	IF xStFct_SetForceDeflection THEN
		IF NOT(xStFct_InitSetForceDeflection) THEN
			IF NOT(ptrTCylToolDeflection^.T_CtrleCyl.xExecute) AND ptrTCylToolDeflection^.T_CtrleCyl.xDone THEN
				xStFct_InitSetForceDeflection:=TRUE;
				ptrTCylToolDeflection^.T_CtrleCyl.iFunction:=4;
				ptrTCylToolDeflection^.T_CtrleCyl.xExecute:=TRUE;
			END_IF;
		END_IF;
		IF NOT(ptrTCylToolDeflection^.T_CtrleCyl.xExecute) AND ptrTCylToolDeflection^.T_CtrleCyl.xDone AND xStFct_InitSetForceDeflection THEN
			xStFct_InitSetForceDeflection:=FALSE;
			xStFct_SetForceDeflection:=FALSE;
		END_IF;
	END_IF;
END_IF;
END_ACTION
ACTION StationFunction_Ctrl_Stop:
IF xStFct_TmpStop AND NOT(xStFct_SetEnd) THEN
	CASE iStFct_TmpStopStep OF
		1:	IF gxHardwareOFF OR gxAxisOFF THEN
				iStFct_TmpStopStep:=9;
				RETURN;
			END_IF;
			IF (NOT(ptrTAxisZ^.T_CtrleSingle.xNotMoving) OR NOT(ptrTAxisZ^.T_CtrleSingle.xDone)) AND
			     NOT((ptrTAxisZ^.T_CtrleSingle.iFunction = 5) AND NOT(ptrTAxisZ^.T_CtrleSingle.xDone)) THEN
				ptrTAxisZ^.T_CtrleSingle.iFunction:=5;
				ptrTAxisZ^.T_CtrleSingle.xExecute:=TRUE;
			END_IF;
			IF (iStationFunctionNr = 5) AND ((iStFct_StepPrc = 3) OR (iStFct_StepPrc = 40)) THEN
				IF (T_Station_Parameter.T_StProcess.iWorkControlType > 1) THEN
					T_Z_St1_Ctrle.diVelocityCommandValue:=0;
					gxZAxisVelocityCtrlActive:=TRUE;
					ptrTAxisZ^.T_CtrleSingle.iFunction:=5;
					ptrTAxisZ^.T_CtrleSingle.xExecute:=TRUE;
				END_IF;
			END_IF;
			IF (NOT(ptrTAxisS^.T_CtrleSingle.xNotMoving) OR NOT(ptrTAxisS^.T_CtrleSingle.xDone)) AND
			     NOT((ptrTAxisS^.T_CtrleSingle.iFunction = 5) AND NOT(ptrTAxisS^.T_CtrleSingle.xDone)) THEN
				ptrTAxisS^.T_CtrleSingle.iFunction:=5;
				ptrTAxisS^.T_CtrleSingle.xExecute:=TRUE;
			END_IF;
			iStFct_TmpStopStep:=iStFct_TmpStopStep + 1;
			T_Station_Work.TCtrlOnlineChange.xLockChange_Z_WorkSpeedForward:=TRUE;
			T_Station_Work.TCtrlOnlineChange.xLockChange_Z_WorkSpeedBackward:=TRUE;
			QxCoolant_St1:=FALSE;
			QxFastStrokeOn_St1:=FALSE;
		2:	IF ptrTAxisZ^.T_CtrleSingle.xNotMoving AND ptrTAxisS^.T_CtrleSingle.xNotMoving AND NOT(gxZAxisVelocityCtrlActive) THEN
				iStFct_TmpStopStep:=iStFct_TmpStopStep + 1;
			ELSE
				IF NOT(gxZAxisVelocityCtrlActive) THEN
					iStFct_TmpStopStep:=1;
				ELSE
					iStFct_TmpStopStep:=10;
				END_IF;
			END_IF;
		3:	IF TRUE THEN
				IF (iStationFunctionNr = 4) OR (iStationFunctionNr = 5) THEN
					iStFct_TmpStopStep:=iStFct_TmpStopStep + 1;
				ELSE
					iStFct_TmpStopStep:=iStFct_TmpStopStep + 6;
				END_IF;
			END_IF;
		4:	T_Station_Work.THWWorkStation.TCtrlWork.xWorkingFinished:=TRUE;
			IF (T_Station_Work.THWWorkStation.TCtrlWork.bPartQuality = 7) THEN
				T_Station_Work.THWWorkStation.TCtrlWork.bPartQuality:=8;	(* < Bearb. abgbr. > *)
			END_IF;
			ptrTAxisZ^.T_CtrleSingle.iFunction:=7;	(* Absolut Bewegung *)
			ptrTAxisZ^.T_CtrleSingle.lrPosition:=grZ_LoadPos;	(* AxisSlide auf LadePosition setzen *)
			ptrTAxisZ^.T_CtrleSingle.lrVelocity:=rOutfeedStrokeAxisSpeed;
			ptrTAxisZ^.T_CtrleSingle.xExecute:=TRUE;
			(* Spindel mit Ausfahrgeschwindigkeit *)
			IF ptrTAxisS^.T_CtrleSingle.xNotMoving THEN
				ptrTAxisS^.T_CtrleSingle.iFunction:=6;	(* Move Velocity *)
			ELSE
				ptrTAxisS^.T_CtrleSingle.iFunction:=12;	(* Move Velocity *)
			END_IF;
			ptrTAxisS^.T_CtrleSingle.lrVelocity:=T_Station_Parameter.T_StProcess.rOutfeedSpindleSpeed;
			ptrTAxisS^.T_CtrleSingle.xExecute:=TRUE;
			IF NOT(ptrTAxisBubbler^.T_CtrleDCAxis.xNotMoving) THEN
				(* Abstreifer ZU *)
				QxCylStripperClose_St1:=TRUE;
				QxCylStripperOpen_St1:=FALSE;
			END_IF
			iStFct_TmpStopStep:=iStFct_TmpStopStep + 1;
		5:	IF NOT(ptrTAxisZ^.T_CtrleSingle.xExecute) AND ptrTAxisZ^.T_CtrleSingle.xDone AND
			     NOT(ptrTAxisS^.T_CtrleSingle.xExecute) AND ptrTAxisS^.T_CtrleSingle.xDone THEN
				iStFct_TmpStopStep:=iStFct_TmpStopStep + 1;
			END_IF;
		6:	IF TRUE THEN
				iStFct_TmpStopStep:=iStFct_TmpStopStep + 1;
			END_IF;
		7:	iStFct_TmpStopStep:=iStFct_TmpStopStep + 1;
		8:	IF NOT(ptrTAxisZ^.T_CtrleSingle.xExecute) AND ptrTAxisZ^.T_CtrleSingle.xDone THEN
				iStFct_TmpStopStep:=iStFct_TmpStopStep + 1;
			END_IF;
		9:	IF TRUE THEN
				xStFct_TmpStop:=FALSE;
				iStFct_TmpStopStep:=1;
				xStFct_SetEnd:=TRUE;
				(* Abstreifer AUF *)
				QxCylStripperClose_St1:=FALSE;
				QxCylStripperOpen_St1:=TRUE;
				QxCylWPUnfix_St1:=FALSE;
				gxSuspensionONOFF:=FALSE;
			END_IF;
		10:	IF NOT(ptrTAxisZ^.T_CtrleSingle.xExecute) AND ptrTAxisZ^.T_CtrleSingle.xDone AND ptrTAxisS^.T_CtrleSingle.xNotMoving THEN
				gxZAxisVelocityCtrlActive:=FALSE;
				iStFct_TmpStopStep:=3;
			END_IF;
	END_CASE;
END_IF;
END_ACTION
ACTION StationFunction_Ctrl_ToolSpindle:
IF NOT(xSafetyCircuitOn) THEN
	T_Station_Work.THWWorkStation.TCtrlWork.xWorkStartToolRotation:=FALSE;
	T_Station_Work.THWWorkStation.TCtrlWork.xWorkStopToolRotation:=FALSE;
END_IF;
IF T_Station_Work.THWWorkStation.TCtrlWork.xWorkStartToolRotation AND NOT(T_Station_Work.THWWorkStation.TCtrlWork.xWorkStopToolRotation) THEN
	CASE iStFct_StepStartToolSpindle OF
	1:	IF NOT(xStFct_InitStepStartToolSpindle) THEN
			IF NOT(ptrTAxisS^.T_CtrleSingle.xExecute) AND NOT(ptrTAxisS^.T_CtrleSingle.xPower) AND ptrTAxisS^.T_CtrleSingle.xDone THEN
				xStFct_InitStepStartToolSpindle:=TRUE;
				ptrTAxisS^.T_CtrleSingle.iFunction:=3;	(* Strom einschalten *)
				ptrTAxisS^.T_CtrleSingle.xExecute:=TRUE;
			END_IF;
		END_IF;
		IF NOT(ptrTAxisS^.T_CtrleSingle.xExecute) AND ptrTAxisS^.T_CtrleSingle.xDone AND ptrTAxisS^.T_CtrleSingle.xPower THEN
			xStFct_InitStepStartToolSpindle:=FALSE;
			iStFct_StepStartToolSpindle:=iStFct_StepStartToolSpindle + 1;
		END_IF;
	2:	IF NOT(xStFct_InitStepStartToolSpindle) THEN
			xStFct_InitStepStartToolSpindle:=TRUE;
			(* Neu-->Hier wird die Spindel nicht mehr mittels der Einfädelgeschwindigkeit gestartet, sondern nur direkt über die Stationseinfädelfunktion *)
		END_IF;
		IF NOT(ptrTAxisS^.T_CtrleSingle.xExecute) AND ptrTAxisS^.T_CtrleSingle.xDone THEN
			xStFct_InitStepStartToolSpindle:=FALSE;
			iStFct_StepStartToolSpindle:=iStFct_StepStartToolSpindle + 1;
		END_IF;
	(* Abwarten bis Einfädeln Bearbeitungsfunktion gestartet hat *)
	3:	IF xStartFunction AND (iStationFunctionNr = 4) THEN
			xStFct_InitStepStartToolSpindle:=FALSE;
			iStFct_StepStartToolSpindle:=iStFct_StepStartToolSpindle + 1;
		END_IF;
	(* Abwarten bis Bearbeitungsfunktion beendet hat *)
	4:	IF NOT(xStartFunction) AND (iStationFunctionNr = 5) THEN
			xStFct_InitStepStartToolSpindle:=FALSE;
			iStFct_StepStartToolSpindle:=iStFct_StepStartToolSpindle + 1;	(* Neu-->Spindel wird gestoppt, und dann erst wieder gestartet direkt über die Stationseinfädelfunktion *)
		END_IF;
	5:	IF NOT(xStFct_InitStepStartToolSpindle) THEN
			IF NOT(ptrTAxisS^.T_CtrleSingle.xExecute) AND NOT(ptrTAxisS^.T_CtrleSingle.xNotMoving) AND
			     ptrTAxisS^.T_CtrleSingle.xDone AND (ptrTAxisS^.T_CtrleSingle.iFunction <> 5) THEN
				xStFct_InitStepStartToolSpindle:=TRUE;
				ptrTAxisS^.T_CtrleSingle.iFunction:=5;	(* Rotation stoppen *)
				ptrTAxisS^.T_CtrleSingle.xExecute:=TRUE;
			END_IF;
		END_IF;
		IF NOT(ptrTAxisS^.T_CtrleSingle.xExecute) AND ptrTAxisS^.T_CtrleSingle.xDone AND ptrTAxisS^.T_CtrleSingle.xNotMoving THEN
			xStFct_InitStepStartToolSpindle:=FALSE;
			iStFct_StepStartToolSpindle:=1;
		ELSE
			xStFct_InitStepStartToolSpindle:=FALSE;
		END_IF;
	END_CASE;
ELSE
	iStFct_StepStartToolSpindle:=1;
	xStFct_InitStepStartToolSpindle:=FALSE;
END_IF;
IF T_Station_Work.THWWorkStation.TCtrlWork.xWorkStopToolRotation THEN
	T_Station_Work.THWWorkStation.TCtrlWork.xWorkStartToolRotation:=FALSE;
	CASE iStFct_StepStopToolSpindle OF
	1:	IF NOT(xStFct_InitStepStopToolSpindle) THEN
			IF NOT(ptrTAxisS^.T_CtrleSingle.xExecute) AND NOT(ptrTAxisS^.T_CtrleSingle.xNotMoving) AND
			     ptrTAxisS^.T_CtrleSingle.xDone AND (ptrTAxisS^.T_CtrleSingle.iFunction <> 5) THEN
				xStFct_InitStepStopToolSpindle:=TRUE;
				ptrTAxisS^.T_CtrleSingle.iFunction:=5;	(* Rotation stoppen *)
				ptrTAxisS^.T_CtrleSingle.xExecute:=TRUE;
			END_IF;
		END_IF;
		IF NOT(ptrTAxisS^.T_CtrleSingle.xExecute) AND ptrTAxisS^.T_CtrleSingle.xDone AND ptrTAxisS^.T_CtrleSingle.xNotMoving THEN
			xStFct_InitStepStopToolSpindle:=FALSE;
			iStFct_StepStopToolSpindle:=iStFct_StepStopToolSpindle + 1;
		ELSE
			xStFct_InitStepStopToolSpindle:=FALSE;
		END_IF;
	2:	IF NOT(xStFct_InitStepStopToolSpindle) THEN
			IF NOT(ptrTAxisS^.T_CtrleSingle.xExecute) AND ptrTAxisS^.T_CtrleSingle.xPower AND ptrTAxisS^.T_CtrleSingle.xDone THEN
				xStFct_InitStepStopToolSpindle:=TRUE;
				ptrTAxisS^.T_CtrleSingle.iFunction:=4;	(* Stromlos schalten *)
				ptrTAxisS^.T_CtrleSingle.xExecute:=TRUE;
			END_IF;
		END_IF;
		IF NOT(ptrTAxisS^.T_CtrleSingle.xExecute) AND ptrTAxisS^.T_CtrleSingle.xDone AND NOT(ptrTAxisS^.T_CtrleSingle.xPower) THEN
			xStFct_InitStepStopToolSpindle:=FALSE;
			iStFct_StepStopToolSpindle:=1;
			T_Station_Work.THWWorkStation.TCtrlWork.xWorkStopToolRotation:=FALSE;
		END_IF;
		IF NOT(ptrTAxisS^.T_CtrleSingle.xExecute) AND NOT(ptrTAxisS^.T_CtrleSingle.xNotMoving) THEN
			xStFct_InitStepStopToolSpindle:=FALSE;
			iStFct_StepStopToolSpindle:=1;
		END_IF;
	END_CASE;
ELSE
	iStFct_StepStopToolSpindle:=1;
	xStFct_InitStepStopToolSpindle:=FALSE;
END_IF;
END_ACTION
ACTION StationFunction_Fct_01_Referencing:
(******************************************************************************************************************************************)
(****************************				           Reset Stationsfunktion                                            *****************************)
(******************************************************************************************************************************************)
StationFunction_Ctrl_Reset;
(******************************************************************************************************************************************)
(****************************			        Stationsfunktion Fehler Controller                                    *****************************)
(******************************************************************************************************************************************)
StationFunction_Ctrl_Error;
(******************************************************************************************************************************************)
(****************************				    Stationsfunktion Haupt Controller                               *****************************)
(******************************************************************************************************************************************)
StationFunction_Ctrl_Main;
(******************************************************************************************************************************************)
(****************************			         Stationsfunktion sofort Unterbrechung                           *****************************)
(******************************************************************************************************************************************)
StationFunction_Ctrl_Stop;
(******************************************************************************************************************************************)
(****************************			             Stationsfunktion Hauptablauf                                       *****************************)
(******************************************************************************************************************************************)
IF xStFct_StartMainPrc AND NOT(xStFct_SetEnd) AND NOT(xStFct_HardwareError) AND NOT(xStFct_TmpStop) THEN
	CASE iStFct_StepPrc OF
	1:	xStFct_StartMainPrc:=FALSE;
		xStFct_InitStep:=FALSE;
		iStFct_StepPrc:=1;
	END_CASE;
END_IF;
(******************************************************************************************************************************************)
(****************************			             Stationsfunktion Parallelablauf                                       *****************************)
(******************************************************************************************************************************************)
IF xStFct_StartPrc_Parallel AND NOT(xStFct_SetEnd) AND NOT(xStFct_HardwareError) THEN
	CASE iStFct_StepPrc_Parallel OF
	1:	iStFct_StepPrc_Parallel:=1;
		xStFct_InitStep_Parallel:=FALSE;
		xStFct_StartPrc_Parallel:=FALSE;
	END_CASE;
END_IF;
(******************************************************************************************************************************************)
(****************************				     Stationsfunktion Endprozedur                                    *****************************)
(******************************************************************************************************************************************)
StationFunction_Ctrl_End;
END_ACTION
ACTION StationFunction_Fct_02_InitialState:
(******************************************************************************************************************************************)
(****************************				           Reset Stationsfunktion                                            *****************************)
(******************************************************************************************************************************************)
StationFunction_Ctrl_Reset;
(******************************************************************************************************************************************)
(****************************			        Stationsfunktion Fehler Controller                                    *****************************)
(******************************************************************************************************************************************)
StationFunction_Ctrl_Error;
(******************************************************************************************************************************************)
(****************************				    Stationsfunktion Haupt Controller                               *****************************)
(******************************************************************************************************************************************)
StationFunction_Ctrl_Main;
(******************************************************************************************************************************************)
(****************************			         Stationsfunktion sofort Unterbrechung                           *****************************)
(******************************************************************************************************************************************)
StationFunction_Ctrl_Stop;
(******************************************************************************************************************************************)
(****************************			             Stationsfunktion Hauptablauf                                       *****************************)
(******************************************************************************************************************************************)
IF xStFct_StartMainPrc AND NOT(xStFct_SetEnd) AND NOT(xStFct_HardwareError) AND NOT(xStFct_TmpStop) THEN
(***************************************************************************************************************************************************)
	CASE iStFct_StepPrc OF
	1:	wStFct_Status:=0;
		xBlockCheckLimitSwitch:=TRUE;
		IF gxHardwareOFF OR gxAxisOFF THEN
			iStFct_StepPrc:=12;
			RETURN;
		END_IF;
		IF NOT(ptrTAxisZ^.T_CtrleSingle.xRef) THEN	(* Z Achse muss referenziert sein *)
			xStFct_HardwareError:=TRUE;
			diStFct_TmpErrorNr:=12;	(* Z Achse muss referenziert sein *)
			RETURN;
		END_IF;
		(* Überprüfe alle Positionen der Z Achse *)
		StationFunction_Ctrl_CheckPos_Z;
		IF xStFct_PositionOutRange_Z THEN
			xStFct_HardwareError:=TRUE;
			diStFct_TmpErrorNr:=iStFct_PosErrorNr;
			RETURN;
		END_IF;
		IF NOT(xStFct_InitStep) THEN
			(* Falls Z Achse sich bewegt, dann wird der Motor gestoppt *)
			IF NOT(ptrTAxisZ^.T_CtrleSingle.xExecute) AND NOT(ptrTAxisZ^.T_CtrleSingle.xNotMoving) THEN
				xStFct_InitStep:=TRUE;
				ptrTAxisZ^.T_CtrleSingle.iFunction:=5;
				ptrTAxisZ^.T_CtrleSingle.xExecute:=TRUE;
			END_IF;
		END_IF;
		IF NOT(ptrTAxisZ^.T_CtrleSingle.xExecute) AND ptrTAxisZ^.T_CtrleSingle.xDone AND ptrTAxisZ^.T_CtrleSingle.xNotMoving THEN
			xStFct_StartMainPrc:=FALSE;
			xStFct_InitStep:=FALSE;
			iStFct_StepPrc:=iStFct_StepPrc + 1;
		END_IF;
	2:	IF NOT(xStFct_InitStep) THEN
			(* Falls Z Achse nicht bestromt ist, dann wird der Motorstrom eingeschaltet *)
			IF NOT(ptrTAxisZ^.T_CtrleSingle.xPower) THEN
				xStFct_InitStep:=TRUE;
				ptrTAxisZ^.T_CtrleSingle.iFunction:=3;	(* Strom einschalten *)
				ptrTAxisZ^.T_CtrleSingle.xExecute:=TRUE;
			END_IF;
			QxCylStripperClose_St1:=FALSE;
			QxCylStripperOpen_St1:=TRUE;
			QxCylWPUnfix_St1:=FALSE;
			gxSuspensionONOFF:=FALSE;
		END_IF;
		IF NOT(ptrTAxisZ^.T_CtrleSingle.xExecute) AND ptrTAxisZ^.T_CtrleSingle.xDone AND ptrTAxisZ^.T_CtrleSingle.xPower THEN
			xStFct_StartMainPrc:=FALSE;
			xStFct_InitStep:=FALSE;
			iStFct_StepPrc:=iStFct_StepPrc + 1;
		END_IF;
	3:	IF NOT(xStFct_InitStep) THEN
			xStFct_InitStep:=TRUE;
			(* Zylinder für Auslenkung-->mit Workauslenkkraft *)
			ptrTCylToolDeflection^.T_CtrleCyl.iFunction:=2;
			ptrTCylToolDeflection^.T_Config.tDelayOn:=T#0.4s;
			ptrTCylToolDeflection^.T_CtrleCyl.T_Analog.rForceIn:=T_Station_Parameter.T_OnlineChange.rForceDeflection;
			ptrTCylToolDeflection^.T_CtrleCyl.xExecute:=TRUE;
			(* Zylinder für Drehmoment HC-->mit Schwellwert Startposition *)
			ptrTCylToolTorqueHC^.T_CtrleCyl.iFunction:=2;
			ptrTCylToolTorqueHC^.T_Config.tDelayOn:=T#0.2s;
			ptrTCylToolTorqueHC^.T_CtrleCyl.T_Analog.rForceIn:=T_Station_Parameter.T_OnlineChange.rTorqueLevelHC;
			ptrTCylToolTorqueHC^.T_CtrleCyl.xExecute:=TRUE;
			(* Zylinder für Überlast Drehmoment *)
			ptrTCylToolTorqueOverload^.T_CtrleCyl.iFunction:=2;
			ptrTCylToolTorqueOverload^.T_Config.tDelayOn:=T#0.2s;
			ptrTCylToolTorqueOverload^.T_CtrleCyl.T_Analog.rForceIn:=T_Station_Parameter.T_StProcess.rTorqueLevel_Overload;
			ptrTCylToolTorqueOverload^.T_CtrleCyl.xExecute:=TRUE;
		END_IF;
		IF NOT(ptrTCylToolDeflection^.T_CtrleCyl.xExecute) AND ptrTCylToolDeflection^.T_CtrleCyl.xDone AND
		    NOT(ptrTCylToolTorqueHC^.T_CtrleCyl.xExecute) AND ptrTCylToolTorqueHC^.T_CtrleCyl.xDone AND
		    NOT(ptrTCylToolTorqueOverload^.T_CtrleCyl.xExecute) AND ptrTCylToolTorqueOverload^.T_CtrleCyl.xDone THEN
			xStFct_StartMainPrc:=FALSE;
			xStFct_InitStep:=FALSE;
			IF NOT(ptrTAxisZ^.T_CtrleSingle.xStateHWLimitNeg) AND NOT(ptrTAxisZ^.T_CtrleSingle.xStateHWLimitPos) THEN
				iStFct_StepPrc:=iStFct_StepPrc + 4;
			ELSE
				IF ptrTAxisZ^.T_CtrleSingle.xStateHWLimitNeg AND ptrTAxisZ^.T_CtrleSingle.xStateHWLimitPos THEN
					xStFct_HardwareError:=TRUE;
					diStFct_TmpErrorNr:=3;	(* Z Achse-->Positiver + Negativer HW Endschalter Aktiv *)
					RETURN;
				ELSIF ptrTAxisZ^.T_CtrleSingle.xStateHWLimitNeg THEN
					iStFct_StepPrc:=iStFct_StepPrc + 1;
				ELSE
					iStFct_StepPrc:=iStFct_StepPrc + 2;
				END_IF;
			END_IF;
		END_IF;
	(* Wegfahren vom negativen Endschalters *)
	4:	IF NOT(xStFct_InitStep) THEN
			xStFct_InitStep:=TRUE;
			ptrTAxisZ^.T_CtrleSingle.iFunction:=6;	(* Geschwindigkeits Bewegung *)
			ptrTAxisZ^.T_CtrleSingle.lrVelocity:=1.0;
			ptrTAxisZ^.T_CtrleSingle.xExecute:=TRUE;
		END_IF;
		IF NOT(ptrTAxisZ^.T_CtrleSingle.xStateHWLimitNeg) THEN
			xStFct_StartMainPrc:=FALSE;
			xStFct_InitStep:=FALSE;
			iStFct_StepPrc:=iStFct_StepPrc + 2;
		END_IF;
		IF ptrTAxisZ^.T_CtrleSingle.xStateHWLimitNeg AND ptrTAxisZ^.T_CtrleSingle.xStateHWLimitPos THEN
			xStFct_HardwareError:=TRUE;
			diStFct_TmpErrorNr:=3;	(* Z Achse-->Positiver + Negativer HW Endschalter Aktiv *)
		END_IF;
	(* Wegfahren vom positiven Endschalters *)
	5:	IF NOT(xStFct_InitStep) THEN
			xStFct_InitStep:=TRUE;
			ptrTAxisZ^.T_CtrleSingle.iFunction:=6;	(* Geschwindigkeits Bewegung *)
			ptrTAxisZ^.T_CtrleSingle.lrVelocity:=-1.0;
			ptrTAxisZ^.T_CtrleSingle.xExecute:=TRUE;
		END_IF;
		IF NOT(ptrTAxisZ^.T_CtrleSingle.xStateHWLimitPos) THEN
			xStFct_StartMainPrc:=FALSE;
			xStFct_InitStep:=FALSE;
			iStFct_StepPrc:=iStFct_StepPrc + 1;
		END_IF;
		IF ptrTAxisZ^.T_CtrleSingle.xStateHWLimitNeg AND ptrTAxisZ^.T_CtrleSingle.xStateHWLimitPos THEN
			xStFct_HardwareError:=TRUE;
			diStFct_TmpErrorNr:=3;	(* Z Achse-->Positiver + Negativer HW Endschalter Aktiv *)
		END_IF;
	(* Stoppen der Bewegung *)
	6:	IF NOT(xStFct_InitStep) THEN
			xStFct_InitStep:=TRUE;
			ptrTAxisZ^.T_CtrleSingle.iFunction:=5;
			ptrTAxisZ^.T_CtrleSingle.xExecute:=TRUE;
		END_IF;
		IF NOT(ptrTAxisZ^.T_CtrleSingle.xExecute) AND ptrTAxisZ^.T_CtrleSingle.xDone THEN
			xStFct_StartMainPrc:=FALSE;
			xStFct_InitStep:=FALSE;
			iStFct_StepPrc:=iStFct_StepPrc + 1;
		END_IF;
	(* Aktuatoren in Ausgangslage bringen *)
	7:	IF NOT(xStFct_InitStep) THEN
			xStFct_InitStep:=TRUE;
			xBlockCheckLimitSwitch:=FALSE;
		END_IF;
		IF TRUE THEN
			xStFct_StartMainPrc:=FALSE;
			xStFct_InitStep:=FALSE;
			iStFct_StepPrc:=iStFct_StepPrc + 1;
		END_IF;
	8:	IF NOT(xStFct_InitStep) THEN
			xStFct_InitStep:=TRUE;
			IF (ptrTAxisZ^.T_LiveValue.lrActualPosition > grZ_LoadPos) THEN
				ptrTAxisZ^.T_CtrleSingle.iFunction:=7;	(* Absolut Bewegung *)
				ptrTAxisZ^.T_CtrleSingle.lrPosition:=grZ_LoadPos;	(* AxisSlide auf LadePosition setzen *)
				ptrTAxisZ^.T_CtrleSingle.lrVelocity:=T_Station_Parameter.T_StProcess.rOutfeedStrokeAxisSpeed;
				ptrTAxisZ^.T_CtrleSingle.xExecute:=TRUE;
			END_IF;
		END_IF;
		IF NOT(ptrTAxisZ^.T_CtrleSingle.xExecute) AND ptrTAxisZ^.T_CtrleSingle.xDone THEN
			xStFct_StartMainPrc:=FALSE;
			xStFct_InitStep:=FALSE;
			iStFct_StepPrc:=iStFct_StepPrc + 1;
		END_IF;
	(* Aktuatoren in Ausgangslage bringen *)
	9:	IF NOT(xStFct_InitStep) THEN
			xStFct_InitStep:=TRUE;
		END_IF;
		IF NOT(ptrTAxisZ^.T_CtrleSingle.xExecute) AND ptrTAxisZ^.T_CtrleSingle.xDone THEN
			xStFct_StartMainPrc:=FALSE;
			xStFct_InitStep:=FALSE;
			iStFct_StepPrc:=iStFct_StepPrc + 1;
		END_IF;
	(* Aktuatoren in Ausgangslage bringen *)
	10:	IF NOT(xStFct_InitStep) THEN
			xStFct_InitStep:=TRUE;
		END_IF;
		IF NOT(ptrTAxisZ^.T_CtrleSingle.xExecute) AND ptrTAxisZ^.T_CtrleSingle.xDone THEN
			xStFct_StartMainPrc:=FALSE;
			xStFct_InitStep:=FALSE;
			iStFct_StepPrc:=iStFct_StepPrc + 1;
		END_IF;
	11:	IF NOT(xStFct_InitStep) THEN
			xStFct_InitStep:=TRUE;
		END_IF;
		IF NOT(ptrTAxisZ^.T_CtrleSingle.xExecute) AND ptrTAxisZ^.T_CtrleSingle.xDone THEN
			xStFct_StartMainPrc:=FALSE;
			xStFct_InitStep:=FALSE;
			iStFct_StepPrc:=iStFct_StepPrc + 1;
		END_IF;
	12:	xStFct_StartMainPrc:=FALSE;
		xStFct_InitStep:=FALSE;
		iStFct_StepPrc:=0;
		xStFct_SetEnd:=TRUE;
	END_CASE;
END_IF;
(******************************************************************************************************************************************)
(****************************			             Stationsfunktion Parallelablauf                                       *****************************)
(******************************************************************************************************************************************)
IF xStFct_StartPrc_Parallel AND NOT(xStFct_SetEnd) AND NOT(xStFct_HardwareError) THEN
	CASE iStFct_StepPrc_Parallel OF
	1:	iStFct_StepPrc_Parallel:=1;
		xStFct_InitStep_Parallel:=FALSE;
		xStFct_StartPrc_Parallel:=FALSE;
	END_CASE;
END_IF;
(******************************************************************************************************************************************)
(****************************				     Stationsfunktion Endprozedur                                    *****************************)
(******************************************************************************************************************************************)
StationFunction_Ctrl_End;
END_ACTION
ACTION StationFunction_Fct_03_ToolRotationON:
;(******************************************************************************************************************************************)
(****************************				           Reset Stationsfunktion                                            *****************************)
(******************************************************************************************************************************************)
StationFunction_Ctrl_Reset;
(******************************************************************************************************************************************)
(****************************			        Stationsfunktion Fehler Controller                                    *****************************)
(******************************************************************************************************************************************)
StationFunction_Ctrl_Error;
(******************************************************************************************************************************************)
(****************************				    Stationsfunktion Haupt Controller                               *****************************)
(******************************************************************************************************************************************)
StationFunction_Ctrl_Main;
(******************************************************************************************************************************************)
(****************************			         Stationsfunktion sofort Unterbrechung                           *****************************)
(******************************************************************************************************************************************)
StationFunction_Ctrl_Stop;
(******************************************************************************************************************************************)
(****************************			             Stationsfunktion Hauptablauf                                       *****************************)
(******************************************************************************************************************************************)
IF xStFct_StartMainPrc AND NOT(xStFct_SetEnd) AND NOT(xStFct_HardwareError) AND NOT(xStFct_TmpStop) THEN
	IF T_Station_Work.THWWorkStation.TCtrlWork.xWorkStopToolRotation THEN
		xStFct_StartMainPrc:=FALSE;
		xStFct_InitStep:=FALSE;
		iStFct_StepPrc:=0;
		xStFct_SetEnd:=TRUE;
	END_IF;
	CASE iStFct_StepPrc OF
	1:	IF NOT(xStFct_InitStep) THEN
			(* Falls die Spindel nicht bestromt ist, dann wird der Motorstrom eingeschaltet *)
			IF NOT(ptrTAxisS^.T_CtrleSingle.xPower) THEN
				xStFct_InitStep:=TRUE;
				ptrTAxisS^.T_CtrleSingle.iFunction:=3;	(* Strom einschalten *)
				ptrTAxisS^.T_CtrleSingle.xExecute:=TRUE;
			END_IF;
		END_IF;
		IF NOT(ptrTAxisS^.T_CtrleSingle.xExecute) AND ptrTAxisS^.T_CtrleSingle.xDone AND ptrTAxisS^.T_CtrleSingle.xPower THEN
			xStFct_StartMainPrc:=FALSE;
			xStFct_InitStep:=FALSE;
			iStFct_StepPrc:=iStFct_StepPrc + 1;
		END_IF;
	2:	IF NOT(xStFct_InitStep) THEN
			xStFct_InitStep:=TRUE;
			(* Zylinder für Auslenkung-->mit Workauslenkkraft *)
			ptrTCylToolDeflection^.T_CtrleCyl.iFunction:=2;
			ptrTCylToolDeflection^.T_Config.tDelayOn:=T#0.3s;
			ptrTCylToolDeflection^.T_CtrleCyl.T_Analog.rForceIn:=T_Station_Parameter.T_OnlineChange.rForceDeflection;
			ptrTCylToolDeflection^.T_CtrleCyl.xExecute:=TRUE;
			(* Zylinder für Drehmoment HC-->mit Schwellwert Startposition *)
			ptrTCylToolTorqueHC^.T_CtrleCyl.iFunction:=2;
			ptrTCylToolTorqueHC^.T_Config.tDelayOn:=T#0.2s;
			ptrTCylToolTorqueHC^.T_CtrleCyl.T_Analog.rForceIn:=T_Station_Parameter.T_OnlineChange.rTorqueLevelHC;
			ptrTCylToolTorqueHC^.T_CtrleCyl.xExecute:=TRUE;
			(* Zylinder für Überlast Drehmoment *)
			ptrTCylToolTorqueOverload^.T_CtrleCyl.iFunction:=2;
			ptrTCylToolTorqueOverload^.T_Config.tDelayOn:=T#0.2s;
			ptrTCylToolTorqueOverload^.T_CtrleCyl.T_Analog.rForceIn:=T_Station_Parameter.T_StProcess.rTorqueLevel_Overload;
			ptrTCylToolTorqueOverload^.T_CtrleCyl.xExecute:=TRUE;
			IF ptrTAxisS^.T_CtrleSingle.xNotMoving THEN
				ptrTAxisS^.T_CtrleSingle.iFunction:=6;	(* Move Velocity *)
			ELSE
				ptrTAxisS^.T_CtrleSingle.iFunction:=12;	(* Move Velocity with new velocity *)
			END_IF;
			ptrTAxisS^.T_CtrleSingle.lrVelocity:=T_Station_Parameter.T_OnlineChange.rWorkingSpindleSpeed;
			ptrTAxisS^.T_CtrleSingle.xExecute:=TRUE;
		END_IF;
		IF NOT(ptrTCylToolDeflection^.T_CtrleCyl.xExecute) AND ptrTCylToolDeflection^.T_CtrleCyl.xDone AND
		     NOT(ptrTCylToolTorqueHC^.T_CtrleCyl.xExecute) AND ptrTCylToolTorqueHC^.T_CtrleCyl.xDone AND
		     NOT(ptrTCylToolTorqueOverload^.T_CtrleCyl.xExecute) AND ptrTCylToolTorqueOverload^.T_CtrleCyl.xDone AND
		     NOT(ptrTAxisS^.T_CtrleSingle.xExecute) AND ptrTAxisS^.T_CtrleSingle.xDone AND NOT(ptrTAxisS^.T_CtrleSingle.xNotMoving) AND
		     ptrTAxisS^.T_CtrleSingle.xConstantVel THEN
			xStFct_StartMainPrc:=FALSE;
			xStFct_InitStep:=FALSE;
			iStFct_StepPrc:=0;
			xStFct_SetEnd:=TRUE;
		END_IF;
		IF NOT(ptrTCylToolDeflection^.T_CtrleCyl.xExecute) AND ptrTCylToolDeflection^.T_CtrleCyl.xDone AND
		     NOT(ptrTAxisS^.T_CtrleSingle.xExecute) AND ptrTAxisS^.T_CtrleSingle.xDone AND ptrTAxisS^.T_CtrleSingle.xNotMoving THEN
			xStFct_StartMainPrc:=FALSE;
			xStFct_InitStep:=FALSE;
			iStFct_StepPrc:=1;
		END_IF;
	END_CASE;
END_IF;
(******************************************************************************************************************************************)
(****************************			             Stationsfunktion Parallelablauf                                       *****************************)
(******************************************************************************************************************************************)
IF xStFct_StartPrc_Parallel AND NOT(xStFct_SetEnd) AND NOT(xStFct_HardwareError) THEN
	CASE iStFct_StepPrc_Parallel OF
	1:	iStFct_StepPrc_Parallel:=1;
		xStFct_InitStep_Parallel:=FALSE;
		xStFct_StartPrc_Parallel:=FALSE;
	END_CASE;
END_IF;
(******************************************************************************************************************************************)
(****************************				     Stationsfunktion Endprozedur                                    *****************************)
(******************************************************************************************************************************************)
StationFunction_Ctrl_End;
END_ACTION
ACTION StationFunction_Fct_04_InfeedWorking:
(******************************************************************************************************************************************)
(****************************				           Reset Stationsfunktion                                            *****************************)
(******************************************************************************************************************************************)
StationFunction_Ctrl_Reset;
(******************************************************************************************************************************************)
(****************************			        Stationsfunktion Fehler Controller                                    *****************************)
(******************************************************************************************************************************************)
StationFunction_Ctrl_Error;
(******************************************************************************************************************************************)
(****************************				    Stationsfunktion Haupt Controller                               *****************************)
(******************************************************************************************************************************************)
StationFunction_Ctrl_Main;
(******************************************************************************************************************************************)
(****************************			         Stationsfunktion sofort Unterbrechung                           *****************************)
(******************************************************************************************************************************************)
StationFunction_Ctrl_Stop;
(******************************************************************************************************************************************)
(****************************			             Stationsfunktion Hauptablauf                                       *****************************)
(******************************************************************************************************************************************)
IF xStFct_StartMainPrc AND NOT(xStFct_SetEnd) AND NOT(xStFct_HardwareError) AND NOT(xStFct_TmpStop) THEN
(***************************************************************************************************************************************************)
(* Überwachung Drehmoment Überlast *)
	StationFunction_CheckOverload;
	IF xStFct_Overload_StopProcess THEN
		RETURN;
	END_IF;
(***************************************************************************************************************************************************)
(* Überwachung auf die Axiale Auslenkung *)
	IF xStFct_ToolDeflectionActiv THEN
		IF NOT(ptrTCylToolDeflection^.T_CtrleCyl.xStatePosOn) THEN
			xStFct_ToolDeflectionActiv:=FALSE;
			xStFct_InitAxialSensor:=FALSE;
			xStFct_CheckAxialSensor:=FALSE;
		END_IF;
	END_IF;
	IF (ptrTCylToolDeflection^.T_CtrleCyl.xStatePosOn OR xStFct_CheckAxialSensor) AND NOT(xStFct_ToolDeflectionActiv) THEN
		IF NOT(xStFct_InitAxialSensor) THEN
			xStFct_InitAxialSensor:=TRUE;
			xStFct_CheckAxialSensor:=TRUE;
			lrStFct_ActualPosition:=ptrTAxisZ^.T_LiveValue.lrActualPosition;
		END_IF;
		IF NOT(ptrTCylToolDeflection^.T_CtrleCyl.xStatePosOn) THEN
			xStFct_InitAxialSensor:=FALSE;
			xStFct_CheckAxialSensor:=FALSE;
			xStFct_ToolDeflectionActiv:=FALSE;
		END_IF;
		IF (ABS(ptrTAxisZ^.T_LiveValue.lrActualPosition - lrStFct_ActualPosition) >= T_Station_Parameter.T_StProcess.rDeflectionSensorOffset) AND ptrTCylToolDeflection^.T_CtrleCyl.xStatePosOn THEN
			xStFct_ToolDeflectionActiv:=TRUE;
		END_IF;
	END_IF;
(***************************************************************************************************************************************************)
(* Hauptablauf für die Bearbeitung *)
	CASE iStFct_StepPrc OF
	1:	(* Überprüfmechanismen die bestehen müssen, damit diese Funktion gestartet werden kann *)
		IF gxHardwareOFF OR gxAxisOFF THEN
			iStFct_StepPrc:=9;
			xStFct_InitStep:=FALSE;
			RETURN;
		END_IF;
		gxWP_Analyse_ActiveInfeed:=TRUE;
		IF NOT(ptrTAxisZ^.T_CtrleSingle.xRef) THEN	(* Z Achse muss referenziert sein *)
			xStFct_HardwareError:=TRUE;
			diStFct_TmpErrorNr:=9;	(* Z Achse muss referenziert sein *)
			RETURN;
		END_IF;
		(* Überprüfe alle Positionen der Z Achse *)
		StationFunction_Ctrl_CheckPos_Z;
		IF xStFct_PositionOutRange_Z THEN
			xStFct_HardwareError:=TRUE;
			diStFct_TmpErrorNr:=iStFct_PosErrorNr;
			RETURN;
		END_IF;
		IF (garPositionEndProcCalc[1] > T_Station_Parameter.T_StProcess.rPositionEndMech) THEN
			xStFct_HardwareError:=TRUE;
			diStFct_TmpErrorNr:=12;		(* Hubprozesslänge > Z Mech EndPos *)
			RETURN;
		END_IF;
		IF (garCentringEndProcCalc[1] > T_Station_Parameter.T_StProcess.rPositionEndMech) THEN
			xStFct_HardwareError:=TRUE;
			diStFct_TmpErrorNr:=18;		(* Zentrier EndPos > Z Mech EndPos *)
			RETURN;
		END_IF;
		IF (T_Station_Parameter.T_StProcess.iSparkOutStrokeCount <> 0) AND
		     ((T_Station_Parameter.T_StProcess.rSparkOutStrokeLength + garPositionEndProcCalc[1]) > T_Station_Parameter.T_StProcess.rPositionEndMech) THEN
			xStFct_HardwareError:=TRUE;
			diStFct_TmpErrorNr:=13;		(* Ausfunkhub > Z Mech EndPos *)
			RETURN;
		END_IF;
		IF ptrTCylToolDeflection^.T_CtrleCyl.xStatePosOn THEN
			xStFct_HardwareError:=TRUE;
			diStFct_TmpErrorNr:=25;		(* Beim starten der Bearbeitung darf AuslenkSensor nicht ON sein *)
			RETURN;
		END_IF;
		IF ptrTCylToolTorqueHC^.T_CtrleCyl.xStatePosOn OR ptrTSensorTorque^.T_CtrleCyl.xStatePosOn THEN
			xStFct_HardwareError:=TRUE;
			diStFct_TmpErrorNr:=26;		(* Beim starten der Bearbeitung darf DrehmSensorHC nicht ON sein *)
			RETURN;
		END_IF;
		IF ptrTCylToolTorqueOverload^.T_CtrleCyl.xStatePosOn OR ptrTSensorTorqueOverload^.T_CtrleCyl.xStatePosOn THEN
			xStFct_HardwareError:=TRUE;
			diStFct_TmpErrorNr:=11;		(* Beim starten der Bearbeitung darf DrehmSensorHCÜberlast nicht ON sein *)
			RETURN;
		END_IF;
		iStFct_TmpHCStartPosCounter:=0;
		iStFct_TmpNumberTryInfeed:=0;
		iStFct_StepPrc:=iStFct_StepPrc + 1;
	2:	IF NOT(xStFct_InitStep) THEN
			xStFct_InitStep:=TRUE;
			T_Station_Work.TCtrlOnlineChange.xLockChangeCylToolDeflectionForce:=TRUE;
			IF NOT(ptrTAxisS^.T_CtrleSingle.xPower) THEN
				ptrTAxisS^.T_CtrleSingle.iFunction:=3;	(* Strom einschalten *)
				ptrTAxisS^.T_CtrleSingle.xExecute:=TRUE;
			END_IF;
			(* Zylinder für Auslenkung-->mit Einfädelkraft *)
			ptrTCylToolDeflection^.T_CtrleCyl.iFunction:=2;
			ptrTCylToolDeflection^.T_Config.tDelayOn:=T#0.3s;
			ptrTCylToolDeflection^.T_CtrleCyl.T_Analog.rForceIn:=T_Station_Parameter.T_StProcess.rInfeedForceDeflection;
			ptrTCylToolDeflection^.T_CtrleCyl.xExecute:=TRUE;
			(* Zylinder für Drehmoment HC-->mit Schwellwert Startposition *)
			ptrTCylToolTorqueHC^.T_CtrleCyl.iFunction:=2;
			ptrTCylToolTorqueHC^.T_Config.tDelayOn:=T#0.2s;
			ptrTCylToolTorqueHC^.T_CtrleCyl.T_Analog.rForceIn:=T_Station_Parameter.T_OnlineChange.rTorqueLevelHC;
			ptrTCylToolTorqueHC^.T_CtrleCyl.xExecute:=TRUE;
			(* Zylinder für Überlast Drehmoment *)
			ptrTCylToolTorqueOverload^.T_CtrleCyl.iFunction:=2;
			ptrTCylToolTorqueOverload^.T_Config.tDelayOn:=T#0.2s;
			ptrTCylToolTorqueOverload^.T_CtrleCyl.T_Analog.rForceIn:=T_Station_Parameter.T_StProcess.rTorqueLevel_Overload;
			ptrTCylToolTorqueOverload^.T_CtrleCyl.xExecute:=TRUE;
		END_IF;
		IF NOT(ptrTAxisS^.T_CtrleSingle.xExecute) AND ptrTAxisS^.T_CtrleSingle.xDone AND ptrTAxisS^.T_CtrleSingle.xPower AND
		     NOT(ptrTCylToolDeflection^.T_CtrleCyl.xExecute) AND ptrTCylToolDeflection^.T_CtrleCyl.xDone AND
		     NOT(ptrTCylToolTorqueHC^.T_CtrleCyl.xExecute) AND ptrTCylToolTorqueHC^.T_CtrleCyl.xDone AND
		     NOT(ptrTCylToolTorqueOverload^.T_CtrleCyl.xExecute) AND ptrTCylToolTorqueOverload^.T_CtrleCyl.xDone THEN
			xStFct_StartMainPrc:=FALSE;
			xStFct_InitStep:=FALSE;
			iStFct_StepPrc:=iStFct_StepPrc + 1;
		END_IF;
	(* Einfädelgeschwindigkeit setzen *)
	3:	IF NOT(xStFct_InitStep) THEN
			xStFct_InitStep:=TRUE;
			ptrTAxisZ^.T_CtrleSingle.iFunction:=7;	(* Absolut Bewegung *)
			ptrTAxisZ^.T_CtrleSingle.lrPosition:=grZ_WorkStartPos;	(* Z auf StartPosition setzen *)
			ptrTAxisZ^.T_CtrleSingle.lrVelocity:=T_Station_Parameter.T_StProcess.rInfeedZAxisSpeed;	(* Mit Einfädelgeschwindigkeit *)
			ptrTAxisZ^.T_CtrleSingle.xExecute:=TRUE;
			(* Spindel mit Einfädelgeschwindigkeit *)
			IF ptrTAxisS^.T_CtrleSingle.xNotMoving THEN
				ptrTAxisS^.T_CtrleSingle.iFunction:=6;	(* Move Velocity *)
			ELSE
				ptrTAxisS^.T_CtrleSingle.iFunction:=12;	(* Move Velocity *)
			END_IF;
			ptrTAxisS^.T_CtrleSingle.lrVelocity:=T_Station_Parameter.T_StProcess.rInfeedSpindleSpeed;
			ptrTAxisS^.T_CtrleSingle.xExecute:=TRUE;
		END_IF;
		IF TRUE THEN
			xStFct_StartMainPrc:=FALSE;
			xStFct_InitStep:=FALSE;
			iStFct_StepPrc:=iStFct_StepPrc + 1;
		END_IF;
	(* Überwachung ob Auslenkung während dem Einfädeln eintrifft *)
	4:	IF xStFct_ToolDeflectionActiv AND NOT(xStFct_StopSlide) THEN
			xStFct_StopSlide:=TRUE;
			wStFct_Status:=1;	(* 1 = < Wz Auslenk. Sensor > *)
			IF xProcessDone THEN
				T_Station_Work.THWWorkStation.TCtrlWork.bPartQuality:=5;	(* < niO kein Einf. > *)
			END_IF;
		END_IF;
		IF NOT(ptrTAxisZ^.T_CtrleSingle.xExecute) AND ptrTAxisZ^.T_CtrleSingle.xDone THEN
			(* Wz konnte erfolgreich eingefädelt werden *)
			xStFct_StartMainPrc:=FALSE;
			xStFct_InitStep:=FALSE;
			iStFct_StepPrc:=7;
			RETURN;
		END_IF;
		IF xStFct_StopSlide AND NOT(ptrTAxisZ^.T_CtrleSingle.xExecute) AND NOT(ptrTAxisZ^.T_CtrleSingle.xDone) AND
		    NOT(ptrTAxisZ^.T_CtrleSingle.xNotMoving) AND (ptrTAxisZ^.T_CtrleSingle.iFunction <> 12) THEN
			ptrTAxisZ^.T_CtrleSingle.iFunction:=5;
			ptrTAxisZ^.T_CtrleSingle.xExecute:=TRUE;
			(* init. variable *)
			xStFct_StopSlide:=FALSE;
			iStFct_StepPrc:=iStFct_StepPrc + 1;
			xStFct_InitStep:=FALSE;
		END_IF;
	5:	(* Abwarten bis die HubAchse stillsteht *)
		IF NOT(ptrTAxisZ^.T_CtrleSingle.xExecute) AND ptrTAxisZ^.T_CtrleSingle.xDone THEN
			xStFct_StartMainPrc:=FALSE;
			xStFct_InitStep:=FALSE;
			iStFct_StepPrc:=iStFct_StepPrc + 1;
		END_IF;
	6:	(* Z Achse um einen Offset zurücksetzen *)
		IF NOT(xStFct_InitStep) THEN
			xStFct_InitStep:=TRUE;
			IF ((ptrTAxisZ^.T_LiveValue.lrActualPosition - ABS(T_Station_Parameter.T_StProcess.rInfeedOffsetBackward)) >= grZ_LoadPos) AND NOT(T_Station_Work.THWWorkStation.TCtrlWork.xLastTryInfeed) THEN
				ptrTAxisZ^.T_CtrleSingle.iFunction:=8;
				ptrTAxisZ^.T_CtrleSingle.lrDistance:=T_Station_Parameter.T_StProcess.rInfeedOffsetBackward;
				ptrTAxisZ^.T_CtrleSingle.lrVelocity:=T_Station_Parameter.T_StProcess.rOutfeedStrokeAxisSpeed;
			ELSE
				ptrTAxisZ^.T_CtrleSingle.iFunction:=7;
				ptrTAxisZ^.T_CtrleSingle.lrPosition:=grZ_LoadPos;
				ptrTAxisZ^.T_CtrleSingle.lrVelocity:=T_Station_Parameter.T_StProcess.rOutfeedStrokeAxisSpeed;
			END_IF;
			ptrTAxisZ^.T_CtrleSingle.xExecute:=TRUE;
		END_IF;
		IF NOT(ptrTAxisZ^.T_CtrleSingle.xExecute) AND ptrTAxisZ^.T_CtrleSingle.xDone THEN
			(* Wz konnte nicht eingefädelt werden *)
			wStFct_Status:=99;
			xStFct_StartMainPrc:=FALSE;
			xStFct_InitStep:=FALSE;
			iStFct_StepPrc:=iStFct_StepPrc + 2;
			T_Station_Work.THWWorkStation.TCtrlWork.xLastTryInfeed:=FALSE;
		END_IF;
	7:	xStFct_StartMainPrc:=FALSE;
		xStFct_InitStep:=FALSE;
		(* Bearbeitungsstation steht nun Bereit um mit der Bearbeitung zu starten *)
		wStFct_Status:=0;
		T_Station_Work.THWWorkStation.TCtrlWork.xToolInfeeded:=TRUE;
		iStFct_StepPrc:=iStFct_StepPrc + 1;
		IF xProcessDone THEN
			T_Station_Work.THWWorkStation.TCtrlWork.bPartQuality:=2;	(* < Go No HC > *)
		END_IF;
	8:	xStFct_StartMainPrc:=FALSE;
		xStFct_InitStep:=FALSE;
		iStFct_StepPrc:=0;
		xStFct_SetEnd:=TRUE;
		T_Station_Work.TCtrlOnlineChange.xLockChangeCylToolDeflectionForce:=FALSE;
		IF xProcessDone THEN
			IF (NOT(ptrTAxisS^.T_CtrleSingle.xNotMoving) OR NOT(ptrTAxisS^.T_CtrleSingle.xDone))
			AND NOT((ptrTAxisS^.T_CtrleSingle.iFunction = 5) AND NOT(ptrTAxisS^.T_CtrleSingle.xDone)) AND NOT(ptrTAxisS^.T_CtrleSingle.xErr) THEN
				ptrTAxisS^.T_CtrleSingle.iFunction:=5;
				ptrTAxisS^.T_CtrleSingle.xExecute:=TRUE;
			END_IF;
		END_IF;
	(* Gilt nur für falls HW ausgeschaltet ist *)
	9:	IF NOT(xStFct_InitStep) THEN
			xStFct_InitStep:=TRUE;
			TONWorkTime(IN:=FALSE);
		END_IF;
		TONWorkTime(IN:=TRUE,PT:=T#2.0s);
		IF TONWorkTime.Q THEN
			TONWorkTime(IN:=FALSE);
			T_Station_Work.THWWorkStation.TCtrlWork.xToolInfeeded:=TRUE;
			xStFct_StartMainPrc:=FALSE;
			xStFct_InitStep:=FALSE;
			iStFct_StepPrc:=0;
			xStFct_SetEnd:=TRUE;
			wStFct_Status:=0;
		END_IF;
	END_CASE;
END_IF;
(******************************************************************************************************************************************)
(****************************			             Stationsfunktion Parallelablauf                                       *****************************)
(******************************************************************************************************************************************)

(******************************************************************************************************************************************)
(****************************				     Stationsfunktion Endprozedur                                    *****************************)
(******************************************************************************************************************************************)
StationFunction_Ctrl_End;
END_ACTION
ACTION StationFunction_Fct_05_Working:
(******************************************************************************************************************************************)
(****************************				           Reset Stationsfunktion                                            *****************************)
(******************************************************************************************************************************************)
StationFunction_Ctrl_Reset;
(******************************************************************************************************************************************)
(****************************			        Stationsfunktion Fehler Controller                                    *****************************)
(******************************************************************************************************************************************)
StationFunction_Ctrl_Error;
(******************************************************************************************************************************************)
(****************************				    Stationsfunktion Haupt Controller                               *****************************)
(******************************************************************************************************************************************)
StationFunction_Ctrl_Main;
(******************************************************************************************************************************************)
(****************************			         Stationsfunktion sofort Unterbrechung                           *****************************)
(******************************************************************************************************************************************)
StationFunction_Ctrl_Stop;
(******************************************************************************************************************************************)
(****************************			             Stationsfunktion Hauptablauf                                       *****************************)
(******************************************************************************************************************************************)
IF ((iStFct_StepPrc <> 3) AND (iStFct_StepPrc <> 51)) OR (T_Station_Parameter.T_StProcess.iWorkControlType <= 1) OR xStFct_TmpStop THEN
	T_Z_St1_Ctrle.diVelocityCommandValue:=(T_Z_St1_Ctrle.nOutData2[1] * 65536) + T_Z_St1_Ctrle.nOutData2[0];
END_IF;
(* Überwachung für langsame oder schnelle Geschwindigkeit für das zurückfahren nach dem Prozessende *)
IF (ptrTAxisZ^.T_LiveValue.lrActualPosition > T_Station_Parameter.T_StProcess.rZ1AxisPosSwitchFastVel) AND (T_Station_Parameter.T_StProcess.rZ1AxisPosSwitchFastVel <> 0.0) THEN
	(* Langsame Geschwindigkeit ist aktiviert für das zurückfahren nach dem Prozessende *)
	rOutfeedStrokeAxisSpeed:=T_Station_Parameter.T_StProcess.rOutfeedStrokeAxisSpeedSlow;
ELSE
	rOutfeedStrokeAxisSpeed:=T_Station_Parameter.T_StProcess.rOutfeedStrokeAxisSpeed;
	IF (T_Station_Parameter.T_StProcess.rZ1AxisPosSwitchFastVel <> 0.0) AND NOT(xBlockSetFastVelZAxis) THEN
		IF (ptrTAxisZ^.T_CtrleSingle.lrPosition = grZ_LoadPos) THEN
			IF NOT(ptrTAxisZ^.T_CtrleSingle.xExecute) AND NOT(ptrTAxisZ^.T_CtrleSingle.xNotMoving) AND NOT(ptrTAxisZ^.T_CtrleSingle.xDone) AND NOT(ptrTAxisZ^.T_CtrleSingle.xErr) THEN
				ptrTAxisZ^.T_CtrleSingle.lrVelocity:=rOutfeedStrokeAxisSpeed;
				ptrTAxisZ^.T_CtrleSingle.iFunction:=12;	(* Z Achse kann nun fliegend auf die schnelle Geschwindigkeit umgestellt werden *)
				ptrTAxisZ^.T_CtrleSingle.xExecute:=TRUE;
				xBlockSetFastVelZAxis:=TRUE;
			END_IF;
		END_IF;
	END_IF;
END_IF;
IF T_Station_Work.THWWorkStation.TCtrlWork.xWorkingFinished AND xStFct_StartMainPrc THEN
	(* Aufzeichnung des max Drehmomentes für wenn die Bearbeitung beendet hat und die Achse zurückfährt *)
	IF (rActTorque >= T_Station_Parameter.T_InfoProcess.rTorqueMaxAfterWork) AND (rActTorque <> 0.0) AND (ptrTAxisZ^.T_LiveValue.lrActualPosition <= lrStartRecordMaxTorque) THEN
		T_Station_Parameter.T_InfoProcess.rTorqueMaxAfterWork:=rActTorque;
		T_Station_Parameter.T_InfoProcess.rTorqueMaxAfterWorkZPos:=ptrTAxisZ^.T_LiveValue.lrActualPosition;
	END_IF;
ELSE
	lrStartRecordMaxTorque:=ptrTAxisZ^.T_LiveValue.lrActualPosition + T_Station_Parameter.T_StProcess.rZ1AxisOffsetStartRecordTorque;
END_IF;
IF xStFct_StartMainPrc AND NOT(xStFct_SetEnd) AND NOT(xStFct_HardwareError) AND NOT(xStFct_TmpStop) THEN
	IF T_Station_Work.THWWorkStation.TCtrlWork.xWorkingFinished THEN
		gxWP_Analyse_ActiveWork:=FALSE;
		gxWP_Analyse_ActiveInfeed:=FALSE;
	END_IF;
(***************************************************************************************************************************************************)
(* Abhandlung der Reinigungsduese *)
	StationFunction_Ctrl_CleanNozzle;
(***************************************************************************************************************************************************)
(* Berechnung der Bearbeitungsarbeit *)
	StationFunction_Ctrl_CalcProcWork;
(***************************************************************************************************************************************************)
(* Regler für die Bearbeitung *)
	IF (T_Station_Parameter.T_StProcess.iWorkControlType <= 1) THEN
		StationFunction_Ctrl_Controller_1;
	ELSIF (T_Station_Parameter.T_StProcess.iWorkControlType = 2) THEN
		StationFunction_Ctrl_Controller_2;
	ELSE
		StationFunction_Ctrl_Controller_3;
	END_IF;
	StationFunction_Ctrl_Controller_S;
	StationFunction_Ctrl_Controller_O;
(***************************************************************************************************************************************************)
(* Abhandlung von Progressivhub  *)
	IF T_Station_Parameter.T_StProcess.iWorkControlType <= 1 THEN
		StationFunction_Ctrl_ProgressStrokeType1;
	ELSIF T_Station_Parameter.T_StProcess.iWorkControlType = 3 THEN
		StationFunction_Ctrl_ProgressStrokeType3;
	END_IF;
(***************************************************************************************************************************************************)
(* Abhandlung von Ausfunken  *)
	IF T_Station_Parameter.T_StProcess.iWorkControlType <= 1 THEN
		StationFunction_Ctrl_ProgressStrokeType1;
	ELSIF T_Station_Parameter.T_StProcess.iWorkControlType = 3 THEN
		StationFunction_Ctrl_ProgressStrokeType3;
	END_IF;
(***************************************************************************************************************************************************)
(* Berechnung der Schnittgeschwindigkeit *)
	fbStFct_CalcCuttingSpeed(	rActualPosition:=ptrTAxisZ^.T_LiveValue.lrActualPosition,
								iCountStep:=10,
								xCapturePosition:=xStFct_CapturePosition,
								xReset:=xStFct_ResetCalcCutSpeed);
	T_Station_Work.THWWorkStation.TCtrlWork.rCuttingSpeed:=fbStFct_CalcCuttingSpeed.rCuttingSpeed;
(***************************************************************************************************************************************************)
(* Auffangen des ersten HC *)
	IF NOT(xStFct_TmpActiveFirstHC) THEN
		IF (iStFct_StepPrc = 1) THEN
			T_Station_Work.THWWorkStation.TCtrlWork.rLastFirstContactPosition:=T_Station_Work.THWWorkStation.TCtrlWork.rActualFirstContactPosition;
		END_IF;
		T_Station_Work.THWWorkStation.TCtrlWork.rActualFirstContactPosition:=0.0;
		IF (T_Station_Work.THWWorkStation.TCtrlWork.rLastOverLimitPosition <> 0.0) THEN
			xStFct_TmpActiveFirstHC:=TRUE;
			T_Station_Work.THWWorkStation.TCtrlWork.rActualFirstContactPosition:=T_Station_Work.THWWorkStation.TCtrlWork.rLastOverLimitPosition;
			T_Station_Work.THWWorkStation.TCtrlWork.xWP_Analyse_ReadyToReadData:=TRUE;
		END_IF;
	END_IF;
(***************************************************************************************************************************************************)
(* Überwachung der minimalen Prozesszeit *)
	fbStFct_TONProcessMinTime(IN:=xStFct_StartProcessTimer,PT:=REAL_TO_TIME(T_Station_Parameter.T_StProcess.rProcessMinTime * 1000.0));
	IF fbStFct_TONProcessMinTime.Q THEN
		xStFct_MinTimeProcessReady:=TRUE;
	ELSE
		xStFct_MinTimeProcessReady:=FALSE;
	END_IF;
(***************************************************************************************************************************************************)
(* Überwachung Drehmoment Überlast *)
	StationFunction_CheckOverload;
	IF xStFct_Overload_StopProcess THEN
		RETURN;
	END_IF;
(***************************************************************************************************************************************************)
(* Überwachung der maximalen Prozesszeit *)
	fbStFct_TONProcessMaxTime(IN:=xStFct_StartProcessTimer,PT:=REAL_TO_TIME(T_Station_Parameter.T_StProcess.rProcessMaxTime * 1000.0));
	IF fbStFct_TONProcessMaxTime.Q AND NOT(xStFct_TmpStopProcess) THEN
		xStFct_TmpStopProcess:=TRUE;
	END_IF;
	IF xStFct_TmpStopProcess THEN
		IF NOT(xStFct_InitStopProcess) THEN
			IF ptrTCylToolTorqueHC^.T_CtrleCyl.xStatePosOn OR ptrTSensorTorque^.T_CtrleCyl.xStatePosOn OR xStFct_ToolDeflectionActiv THEN
				xStFct_InitStopProcess:=TRUE;
				iStFct_StopProcess:=1;
			END_IF;
		END_IF;
		IF xStFct_InitStopProcess THEN
			T_Station_Work.THWWorkStation.TCtrlWork.bPartQuality:=4;	(* < niO max Zeit > *)
			T_Station_Work.TCtrlOnlineChange.xLockChange_Z_WorkSpeedForward:=TRUE;
			T_Station_Work.TCtrlOnlineChange.xLockChange_Z_WorkSpeedBackward:=TRUE;
			T_Station_Work.TCtrlOnlineChange.xLockChange_S_WorkSpindleSpeed:=TRUE;
			CASE iStFct_StopProcess OF
				1:	IF (T_Station_Parameter.T_StProcess.iWorkControlType <= 1) THEN
						IF (NOT(ptrTAxisZ^.T_CtrleSingle.xNotMoving) OR NOT(ptrTAxisZ^.T_CtrleSingle.xDone)) AND
				     		    NOT((ptrTAxisZ^.T_CtrleSingle.iFunction = 5) AND NOT(ptrTAxisZ^.T_CtrleSingle.xDone)) THEN
							ptrTAxisZ^.T_CtrleSingle.iFunction:=5;
							ptrTAxisZ^.T_CtrleSingle.xExecute:=TRUE;
							iStFct_StopProcess:=iStFct_StopProcess + 1;
						ELSE
							iStFct_StopProcess:=iStFct_StopProcess + 1;
						END_IF;
					ELSE
						T_Z_St1_Ctrle.diVelocityCommandValue:=0;
						gxZAxisVelocityCtrlActive:=TRUE;
						ptrTAxisZ^.T_CtrleSingle.iFunction:=5;
						ptrTAxisZ^.T_CtrleSingle.xExecute:=TRUE;
						iStFct_StopProcess:=iStFct_StopProcess + 1;
					END_IF;
				2:	IF NOT(ptrTAxisZ^.T_CtrleSingle.xExecute) AND ptrTAxisZ^.T_CtrleSingle.xDone AND NOT(gxZAxisVelocityCtrlActive) THEN
						T_Station_Work.THWWorkStation.TCtrlWork.xWorkingFinished:=TRUE;
						ptrTAxisZ^.T_CtrleSingle.iFunction:=7;	(* Absolut Bewegung *)
						ptrTAxisZ^.T_CtrleSingle.lrPosition:=grZ_LoadPos;	(* AxisSlide auf BearbStartPosition setzen *)
						ptrTAxisZ^.T_CtrleSingle.lrVelocity:=rOutfeedStrokeAxisSpeed;
						ptrTAxisZ^.T_CtrleSingle.xExecute:=TRUE;
						(* Spindel mit Ausfahrgeschwindigkeit *)
						IF ptrTAxisS^.T_CtrleSingle.xNotMoving THEN
							ptrTAxisS^.T_CtrleSingle.iFunction:=6;	(* Move Velocity *)
						ELSE
							ptrTAxisS^.T_CtrleSingle.iFunction:=12;	(* Move Velocity *)
						END_IF;
						ptrTAxisS^.T_CtrleSingle.lrVelocity:=T_Station_Parameter.T_StProcess.rOutfeedSpindleSpeed;
						ptrTAxisS^.T_CtrleSingle.xExecute:=TRUE;
						iStFct_StopProcess:=iStFct_StopProcess + 1;
					ELSE
						IF NOT(gxZAxisVelocityCtrlActive) THEN
							iStFct_StopProcess:=1;
						ELSE
							iStFct_StopProcess:=5;
						END_IF;
					END_IF;
				3:	IF NOT(ptrTAxisZ^.T_CtrleSingle.xExecute) AND ptrTAxisZ^.T_CtrleSingle.xDone AND
		     			     NOT(ptrTAxisS^.T_CtrleSingle.xExecute) AND ptrTAxisS^.T_CtrleSingle.xDone THEN
						ptrTAxisZ^.T_CtrleSingle.iFunction:=7;	(* Absolut Bewegung *)
						ptrTAxisZ^.T_CtrleSingle.lrPosition:=grZ_LoadPos;	(* AxisSlide auf LadePosition setzen *)
						ptrTAxisZ^.T_CtrleSingle.lrVelocity:=rOutfeedStrokeAxisSpeed;
						ptrTAxisZ^.T_CtrleSingle.xExecute:=TRUE;
						iStFct_StopProcess:=iStFct_StopProcess + 1;
					END_IF;
				4:	IF NOT(ptrTAxisZ^.T_CtrleSingle.xExecute) AND ptrTAxisZ^.T_CtrleSingle.xDone THEN
						xStFct_SetEnd:=TRUE;
						IF xProcessDone THEN
							IF (NOT(ptrTAxisS^.T_CtrleSingle.xNotMoving) OR NOT(ptrTAxisS^.T_CtrleSingle.xDone)) AND
							     NOT((ptrTAxisS^.T_CtrleSingle.iFunction = 5) AND NOT(ptrTAxisS^.T_CtrleSingle.xDone)) AND NOT(ptrTAxisS^.T_CtrleSingle.xErr) THEN
								ptrTAxisS^.T_CtrleSingle.iFunction:=5;
								ptrTAxisS^.T_CtrleSingle.xExecute:=TRUE;
							END_IF;
						END_IF;
						RETURN;
						xStFct_TmpStopProcess:=FALSE;
					END_IF;
				5:	IF NOT(ptrTAxisZ^.T_CtrleSingle.xExecute) AND ptrTAxisZ^.T_CtrleSingle.xDone THEN
						gxZAxisVelocityCtrlActive:=FALSE;
						iStFct_StopProcess:=2;
					END_IF;
			END_CASE;
			RETURN;
		END_IF;
	END_IF;
(***************************************************************************************************************************************************)
(* Prozessende Ausfunkprozedur *)
	IF T_Station_Parameter.T_StProcess.iSparkOutController <= 2 THEN
		fbStFct_SparkOutProcess(	lrHubLength:= T_Station_Parameter.T_StProcess.rSparkOutStrokeLength,
								iCountHub:= T_Station_Parameter.T_StProcess.iSparkOutStrokeCount,
								T_Station_Parameter:= T_Station_Parameter,
								xStart:= xStFct_StartSparkOutProcess,
								xReset:= xStFct_ResetSparkOutProcess,
								xToolDeflection:= ptrTCylToolDeflection^.T_CtrleCyl.xStatePosOn OR IxToolDeflection2_St1,
								xToolTorqueHC:=ptrTCylToolTorqueHC^.T_CtrleCyl.xStatePosOn OR ptrTSensorTorque^.T_CtrleCyl.xStatePosOn,
								xToolTorqueSparkOut:=ptrTCylToolTorqueHC^.T_CtrleCyl.xStatePosOn1 OR ptrTSensorTorque^.T_CtrleCyl.xStatePosOn1,
								TCylToolDeflection:=ptrTCylToolDeflection^,
								TAxisZ:= ptrTAxisZ^);
	ELSE
		StationFunction_Ctrl_SparkOutType3;
	END_IF
(***************************************************************************************************************************************************)
(* Überwachung auf die Axiale Auslenkung *)
	IF xStFct_ToolDeflectionActiv THEN
		IF NOT(ptrTCylToolDeflection^.T_CtrleCyl.xStatePosOn) AND NOT(IxToolDeflection2_St1) THEN
			xStFct_ToolDeflectionActiv:=FALSE;
			xStFct_InitAxialSensor:=FALSE;
			xStFct_CheckAxialSensor:=FALSE;
		END_IF;
	END_IF;
	IF (ptrTCylToolDeflection^.T_CtrleCyl.xStatePosOn OR IxToolDeflection2_St1 OR xStFct_CheckAxialSensor) AND NOT(xStFct_ToolDeflectionActiv) THEN
		IF NOT(xStFct_InitAxialSensor) THEN
			xStFct_InitAxialSensor:=TRUE;
			xStFct_CheckAxialSensor:=TRUE;
			lrStFct_ActualPosition:=ptrTAxisZ^.T_LiveValue.lrActualPosition;
		END_IF;
		IF NOT(ptrTCylToolDeflection^.T_CtrleCyl.xStatePosOn) AND NOT(IxToolDeflection2_St1) THEN
			xStFct_InitAxialSensor:=FALSE;
			xStFct_CheckAxialSensor:=FALSE;
			xStFct_ToolDeflectionActiv:=FALSE;
		END_IF;
		IF (ABS(ptrTAxisZ^.T_LiveValue.lrActualPosition - lrStFct_ActualPosition) >= T_Station_Parameter.T_StProcess.rDeflectionSensorOffset) AND (ptrTCylToolDeflection^.T_CtrleCyl.xStatePosOn OR IxToolDeflection2_St1) THEN
			xStFct_ToolDeflectionActiv:=TRUE;
		END_IF;
	END_IF;
(***************************************************************************************************************************************************)
	IF (T_Station_Parameter.T_StProcess.iWorkControlType <= 1) OR (T_Station_Parameter.T_StProcess.iWorkControlType = 2) THEN
		TONWaitReady(IN:=ptrTAxisZ^.T_CtrleSingle.xMovingForward AND ptrTAxisZ^.T_CtrleSingle.xConstantVel,PT:=T#0.02s);
	ELSE
		TONWaitReady(IN:=(iStFct_StepPrc = 3) AND NOT(xStFct_StopSlide) AND (ptrTAxisZ^.T_LiveValue.lrActualVelocity <= T_Station_Parameter.T_StProcess.rSpeedZAxisForBackward),PT:=T#0.1s);
	END_IF;
(* Hauptablauf für die Bearbeitung *)
	CASE iStFct_StepPrc OF
	1:	xEndPosReachZylindricalProcess:=FALSE;
		IF gxHardwareOFF OR gxAxisOFF THEN
			IF (garPositionEndProcCalc[1] > T_Station_Parameter.T_StProcess.rPositionEndProcMaxInc) AND (T_Station_Parameter.T_StProcess.xPositionEndProcIncOnOff OR gxProcessCylindricalAreaActive) THEN
				xStFct_HardwareError:=TRUE;
				diStFct_TmpErrorNr:=17;		(* Z Bearb EndPos Berechn. > Z Bearb EndPos Max *)
				RETURN;
			END_IF;
			IF (garCentringEndProcCalc[1] > T_Station_Parameter.T_StProcess.rPositionEndProcMaxInc) AND T_Station_Parameter.T_StProcess.xCentringEndProcIncOnOff THEN
				xStFct_HardwareError:=TRUE;
				diStFct_TmpErrorNr:=19;			(* Z ZentrierPos berechn. > Z Bearb EndPos Max *)
				RETURN;
			END_IF;
			gxWP_Analyse_ActiveWork:=TRUE;
			xStFct_StartMainPrc:=FALSE;
			xStFct_InitStep:=FALSE;
			iStFct_StepPrc:=14;
			RETURN;
		END_IF;
		gxWP_Analyse_ActiveWork:=TRUE;
		(* Überprüfmechanismen die bestehen müssen, damit diese Funktion gestartet werden kann *)
		IF NOT(ptrTAxisZ^.T_CtrleSingle.xRef) THEN	(* Z Achse muss referenziert sein *)
			xStFct_HardwareError:=TRUE;
			diStFct_TmpErrorNr:=9;	(* Z Achse muss referenziert sein *)
			RETURN;
		END_IF;
		(* Überprüfe alle Positionen der Z Achse *)
		StationFunction_Ctrl_CheckPos_Z;
		IF xStFct_PositionOutRange_Z THEN
			xStFct_HardwareError:=TRUE;
			diStFct_TmpErrorNr:=iStFct_PosErrorNr;
			RETURN;
		END_IF;
		IF (garPositionEndProcCalc[1] > T_Station_Parameter.T_StProcess.rPositionEndMech) THEN
			xStFct_HardwareError:=TRUE;
			diStFct_TmpErrorNr:=12;		(* Hubprozesslänge > Z Mech EndPos *)
			RETURN;
		END_IF;
		IF (garCentringEndProcCalc[1] > T_Station_Parameter.T_StProcess.rPositionEndMech) THEN
			xStFct_HardwareError:=TRUE;
			diStFct_TmpErrorNr:=18;		(* Zentrier EndPos > Z Mech EndPos *)
			RETURN;
		END_IF;
		IF (garPositionEndProcCalc[1] > T_Station_Parameter.T_StProcess.rPositionEndProcMaxInc) AND (T_Station_Parameter.T_StProcess.xPositionEndProcIncOnOff OR gxProcessCylindricalAreaActive) THEN
			xStFct_HardwareError:=TRUE;
			diStFct_TmpErrorNr:=17;		(* Z Bearb EndPos Berechn. > Z Bearb EndPos Max *)
			RETURN;
		END_IF;
		IF (garCentringEndProcCalc[1] > T_Station_Parameter.T_StProcess.rPositionEndProcMaxInc) AND T_Station_Parameter.T_StProcess.xCentringEndProcIncOnOff THEN
			xStFct_HardwareError:=TRUE;
			diStFct_TmpErrorNr:=19;			(* Z ZentrierPos berechn. > Z Bearb EndPos Max *)
			RETURN;
		END_IF;
		IF (T_Station_Parameter.T_StProcess.iSparkOutStrokeCount <> 0) AND
		     ((T_Station_Parameter.T_StProcess.rSparkOutStrokeLength + garPositionEndProcCalc[1]) > T_Station_Parameter.T_StProcess.rPositionEndMech) THEN
			xStFct_HardwareError:=TRUE;
			diStFct_TmpErrorNr:=13;		(* Ausfunkhub > Z Mech EndPos *)
			RETURN;
		END_IF;
		IF ptrTCylToolDeflection^.T_CtrleCyl.xStatePosOn OR IxToolDeflection2_St1 THEN
			xStFct_HardwareError:=TRUE;
			diStFct_TmpErrorNr:=25;		(* Beim starten der Bearbeitung darf AuslenkSensor nicht ON sein *)
			RETURN;
		END_IF;
		IF ptrTCylToolTorqueHC^.T_CtrleCyl.xStatePosOn OR ptrTSensorTorque^.T_CtrleCyl.xStatePosOn THEN
			xStFct_HardwareError:=TRUE;
			diStFct_TmpErrorNr:=26;		(* Beim starten der Bearbeitung darf DrehmSensorHC nicht ON sein *)
			RETURN;
		END_IF;
		IF ptrTCylToolTorqueOverload^.T_CtrleCyl.xStatePosOn OR ptrTSensorTorqueOverload^.T_CtrleCyl.xStatePosOn THEN
			xStFct_HardwareError:=TRUE;
			diStFct_TmpErrorNr:=11;		(* Beim starten der Bearbeitung darf DrehmSensorHCÜberlast nicht ON sein *)
			RETURN;
		END_IF;
		(* Überprüfe ob Wz im Wstk eingefädelt ist *)
		IF NOT(ptrTAxisZ^.T_LiveValue.lrActualPosition >= (grZ_WorkStartPos - 0.1)) THEN
			xStFct_HardwareError:=TRUE;
			diStFct_TmpErrorNr:=14;		(* Werkzeug ist nicht im Werkstück eingefädelt *)
			RETURN;
		END_IF;
		(* Zylinder für Auslenkung-->mit Bearbeitungskraft *)
		ptrTCylToolDeflection^.T_CtrleCyl.iFunction:=2;
		ptrTCylToolDeflection^.T_Config.tDelayOn:=T#0.3s;
		ptrTCylToolDeflection^.T_CtrleCyl.T_Analog.rForceIn:=T_Station_Parameter.T_OnlineChange.rForceDeflection;
		ptrTCylToolDeflection^.T_CtrleCyl.xExecute:=TRUE;
		(* Zylinder für Drehmoment HC-->mit Schwellwert Startposition *)
		ptrTCylToolTorqueHC^.T_CtrleCyl.iFunction:=2;
		ptrTCylToolTorqueHC^.T_Config.tDelayOn:=T#0.2s;
		ptrTCylToolTorqueHC^.T_CtrleCyl.T_Analog.rForceIn:=T_Station_Parameter.T_OnlineChange.rTorqueLevelHC;
		ptrTCylToolTorqueHC^.T_CtrleCyl.xExecute:=TRUE;
		(* Zylinder für Überlast Drehmoment *)
		ptrTCylToolTorqueOverload^.T_CtrleCyl.iFunction:=2;
		ptrTCylToolTorqueOverload^.T_Config.tDelayOn:=T#0.2s;
		ptrTCylToolTorqueOverload^.T_CtrleCyl.T_Analog.rForceIn:=T_Station_Parameter.T_StProcess.rTorqueLevel_Overload;
		ptrTCylToolTorqueOverload^.T_CtrleCyl.xExecute:=TRUE;
		iStFct_TmpHCStartPosCounter:=0;
		iStFct_TmpNumberTryInfeed:=0;
		iStFct_StepPrc:=iStFct_StepPrc + 1;
		IF NOT(ptrTAxisS^.T_CtrleSingle.xPower) THEN
			ptrTAxisS^.T_CtrleSingle.iFunction:=3;	(* Strom einschalten *)
			ptrTAxisS^.T_CtrleSingle.xExecute:=TRUE;
		END_IF;
	2:	IF NOT(ptrTAxisS^.T_CtrleSingle.xExecute) AND ptrTAxisS^.T_CtrleSingle.xDone AND ptrTAxisS^.T_CtrleSingle.xPower THEN
			IF NOT(xStFct_InitStep) THEN
				xStFct_InitStep:=TRUE;
				IF (T_Station_Parameter.T_StProcess.iWorkControlType <= 1) THEN
					ptrTAxisZ^.T_CtrleSingle.iFunction:=7;	(* Absolut Bewegung *)
					IF NOT(gxProcessCylindricalAreaActive) THEN
						ptrTAxisZ^.T_CtrleSingle.lrPosition:=garPositionEndProcCalc[1];	(* AxisSlide auf EndPosition setzen *)
					ELSE
						(* Das ist der neue Ablauf wo man einen Zylindrische Position definieren kann und aber dieser Position wenn das Drehmoment einem definierten Schwellwert unterschritten wird, dann ist dies das Prozessende. Wird aber diese unten übergebene Position erreicht, dann wertet es als Fehler *)
						ptrTAxisZ^.T_CtrleSingle.lrPosition:=T_Station_Parameter.T_StProcess.rPositionEndProcMaxInc;
					END_IF;
					ptrTAxisZ^.T_CtrleSingle.lrVelocity:=T_Station_Parameter.T_OnlineChange.rWorkingSpeedForward;
					ptrTAxisZ^.T_CtrleSingle.xExecute:=TRUE;
				END_IF;
				IF ptrTAxisS^.T_CtrleSingle.xNotMoving THEN
					ptrTAxisS^.T_CtrleSingle.iFunction:=6;	(* Move Velocity *)
				ELSE
					ptrTAxisS^.T_CtrleSingle.iFunction:=12;	(* Move Velocity *)
				END_IF;
				ptrTAxisS^.T_CtrleSingle.lrVelocity:=T_Station_Parameter.T_OnlineChange.rWorkingSpindleSpeed;
				ptrTAxisS^.T_CtrleSingle.xExecute:=TRUE;
				xStFct_StartProcessTimer:=TRUE;	(*Min und Max Timer starten*)
				T_Station_Work.THWWorkStation.TCtrlWork.xWorkingStarted:=TRUE;
				IF (T_Station_Parameter.T_StProcess.rWorkingSpeedOscillation > 0.0) THEN
					QxFastStrokeOn_St1:=TRUE;
					QiAFastStroke:=REAL_TO_INT(32757 / 50.0 * T_Station_Parameter.T_StProcess.rWorkingSpeedOscillation);		(* 32767digits / 50Hz * Param Hz *)
				ELSE
					QxFastStrokeOn_St1:=FALSE;
					QiAFastStroke:=0;
				END_IF;
			END_IF;
			IF (T_Station_Parameter.T_StProcess.iWorkControlType <= 1) THEN
				IF NOT(ptrTAxisZ^.T_CtrleSingle.xExecute) AND (NOT(ptrTAxisZ^.T_CtrleSingle.xDone) OR ptrTAxisZ^.T_CtrleSingle.xNotMoving) AND
				     NOT(ptrTAxisS^.T_CtrleSingle.xExecute) AND ptrTAxisS^.T_CtrleSingle.xDone THEN
					T_Station_Work.TCtrlOnlineChange.xLockChange_S_WorkSpindleSpeed:=FALSE;
					xStFct_StartMainPrc:=FALSE;
					xStFct_InitStep:=FALSE;
					iStFct_StepPrc:=iStFct_StepPrc + 1;
					RETURN;
				END_IF;
				(* Überwachung falls während der Zeit dass die Bearbeitungsparameter übergeben werden ein HC eintreffen sollte *)
				IF xStFct_ToolDeflectionActiv OR ptrTCylToolTorqueHC^.T_CtrleCyl.xStatePosOn OR ptrTSensorTorque^.T_CtrleCyl.xStatePosOn THEN
					T_Station_Work.TCtrlOnlineChange.xLockChange_S_WorkSpindleSpeed:=FALSE;
					xStFct_StartMainPrc:=FALSE;
					xStFct_InitStep:=FALSE;
					iStFct_StepPrc:=iStFct_StepPrc + 1;
				END_IF;
			ELSE
				IF  NOT(ptrTAxisS^.T_CtrleSingle.xExecute) AND ptrTAxisS^.T_CtrleSingle.xDone THEN
					xStFct_StartMainPrc:=FALSE;
					xStFct_InitStep:=FALSE;
					iStFct_StepPrc:=iStFct_StepPrc + 1;
				END_IF;
			END_IF;
		END_IF;
	3:	(* Bearbeitungsprozess ist nun Aktiv-->Wstk wird effektiv bearbeitet *)
		T_Station_Work.TCtrlOnlineChange.xLockChange_Z_WorkSpeedForward:=FALSE;	(* OnlineChange Parameter kann für die HubAchse Vorwärtsgeschw. aktiviert werden *)
		IF gxProcessCylindricalAreaActive AND NOT(xEndPosReachZylindricalProcess) THEN
			(* Beim neuen Ablauf sobald der Zylindrische Bereich erreicht wird, dann muss die Überwachung des Drehmomentschwellwertes aktiviert werden und wenn dieser unterschritten wird, dann gilt dies als EndPosition der Bearbeitung *)
			IF (ptrTAxisZ^.T_LiveValue.lrActualPosition >= garPositionEndProcCalc[1]) THEN		(* Beachte die Position garPositionEndProcCalc[1] bei neuem Ablauf ist mit dem Zylindrischen Bereich verknüpft inklusiv Inkrementierung *)
				IF (T_Station_Work.THWWorkStation.TCtrlWork.iProgressBar_Torque < T_Station_Parameter.T_StProcess.rZMinThresholdTroqueEndProcess) THEN
					(* Man befindet sich im zylindrischen Bereich und das Drehmoment wurde vom vorgegebenen Schwellwert unterschritten und gilt als Prozessende *)
					IF (T_Station_Parameter.T_StProcess.iWorkControlType <= 1) THEN
						IF (NOT(ptrTAxisZ^.T_CtrleSingle.xExecute) AND NOT(ptrTAxisZ^.T_CtrleSingle.xDone) AND NOT(ptrTAxisZ^.T_CtrleSingle.xNotMoving) AND (ptrTAxisZ^.T_CtrleSingle.iFunction <> 12)) THEN
							ptrTAxisZ^.T_CtrleSingle.iFunction:=5;
							ptrTAxisZ^.T_CtrleSingle.xExecute:=TRUE;
							xEndPosReachZylindricalProcess:=TRUE;
						END_IF;
					ELSE
						xEndPosReachZylindricalProcess:=TRUE;
					END_IF;
					T_Station_Parameter.T_StProcess.rZPositionCylindricalAreaStop:=ptrTAxisZ^.T_LiveValue.lrActualPosition;
					T_ExchgParam.T_StationCommon.T_Param_StationWork.T_StProcess.rZPositionCylindricalAreaStop:=T_Station_Parameter.T_StProcess.rZPositionCylindricalAreaStop;
				END_IF;
			END_IF;
		END_IF;
		IF (T_Station_Parameter.T_StProcess.iWorkControlType <> 2) THEN
			IF xStFct_ToolDeflectionActiv AND NOT(ptrTCylToolTorqueHC^.T_CtrleCyl.xStatePosOn) AND NOT(ptrTSensorTorque^.T_CtrleCyl.xStatePosOn) AND NOT(xStFct_StopSlide) AND NOT(xEndPosReachZylindricalProcess) THEN
				xStFct_StopSlide:=TRUE;
				wStFct_Status:=1;	(* 1 = < Wz Auslenk. Sensor > *)
				T_Station_Work.THWWorkStation.TCtrlWork.xDeflectionLastHC:=TRUE;
				T_Station_Work.THWWorkStation.TCtrlWork.xTorqueLastHC:=FALSE;
			END_IF;
			IF (ptrTCylToolTorqueHC^.T_CtrleCyl.xStatePosOn OR ptrTSensorTorque^.T_CtrleCyl.xStatePosOn) AND NOT(xStFct_ToolDeflectionActiv) AND NOT(xStFct_StopSlide) AND NOT(xEndPosReachZylindricalProcess) THEN
				xStFct_StopSlide:=TRUE;
				wStFct_Status:=2;	(* 2 = < Wz Drehmom. HC> *)
				T_Station_Work.THWWorkStation.TCtrlWork.xDeflectionLastHC:=FALSE;
				T_Station_Work.THWWorkStation.TCtrlWork.xTorqueLastHC:=TRUE;
			END_IF
			IF xStFct_ToolDeflectionActiv AND (ptrTCylToolTorqueHC^.T_CtrleCyl.xStatePosOn OR  ptrTSensorTorque^.T_CtrleCyl.xStatePosOn) AND NOT(xStFct_StopSlide) AND NOT(xEndPosReachZylindricalProcess) THEN
				xStFct_StopSlide:=TRUE;
				wStFct_Status:=3;	(* 3 = < Wz Auslenk.+Wz Drehm.HC > *)
				T_Station_Work.THWWorkStation.TCtrlWork.xDeflectionLastHC:=TRUE;
				T_Station_Work.THWWorkStation.TCtrlWork.xTorqueLastHC:=TRUE;
			END_IF;
			IF (ptrTAxisZ^.T_LiveValue.lrActualVelocity <= T_Station_Parameter.T_StProcess.rSpeedZAxisForBackward) AND NOT(xStFct_StopSlide) AND TONWaitReady.Q AND NOT(xEndPosReachZylindricalProcess) THEN
				xStFct_StopSlide:=TRUE;
				wStFct_Status:=4;	(* 4 = < Z min Geschw. > *)
				T_Station_Work.THWWorkStation.TCtrlWork.xDeflectionLastHC:=TRUE;
				T_Station_Work.THWWorkStation.TCtrlWork.xTorqueLastHC:=TRUE;
			END_IF;
		ELSE
			IF xStFct_ToolDeflectionActiv AND NOT(ptrTCylToolTorqueHC^.T_CtrleCyl.xStatePosOn) AND NOT(ptrTSensorTorque^.T_CtrleCyl.xStatePosOn) AND NOT(xStFct_StopSlide) AND NOT(xEndPosReachZylindricalProcess) THEN
				xStFct_StopSlide:=TRUE;
				wStFct_Status:=1;	(* 1 = < Wz Auslenk. Sensor > *)
				T_Station_Work.THWWorkStation.TCtrlWork.xDeflectionLastHC:=TRUE;
				T_Station_Work.THWWorkStation.TCtrlWork.xTorqueLastHC:=FALSE;
			END_IF;
		END_IF;
		IF xStFct_StopSlide AND ((NOT(ptrTAxisZ^.T_CtrleSingle.xExecute) AND NOT(ptrTAxisZ^.T_CtrleSingle.xDone) AND
		    NOT(ptrTAxisZ^.T_CtrleSingle.xNotMoving) AND (ptrTAxisZ^.T_CtrleSingle.iFunction <> 12)) OR
 		    (T_Station_Parameter.T_StProcess.iWorkControlType = 2) OR (T_Station_Parameter.T_StProcess.iWorkControlType = 3)) THEN
			T_Station_Work.TCtrlOnlineChange.xLockChange_Z_WorkSpeedForward:=TRUE;
			IF (T_Station_Parameter.T_StProcess.iWorkControlType <= 1) THEN
				ptrTAxisZ^.T_CtrleSingle.iFunction:=5;
				ptrTAxisZ^.T_CtrleSingle.xExecute:=TRUE;
			END_IF;
			rStFct_SetZHCPosition:=ptrTAxisZ^.T_LiveValue.lrActualPosition;
			xStFct_CapturePosition:=TRUE;	(* Berechnung der Schnittgeschwindigkeit *)
			xStFct_HCActivated:=TRUE;	(* Überwachung für das Einfressen des Wz im Wstk *)
			IF NOT(xStFct_ForceHC) THEN
				IF (rStFct_TmpDiffOverLimitPosition <> 0) THEN
					T_Station_Work.THWWorkStation.TCtrlWork.rDiffOverLimitPosition:=ptrTAxisZ^.T_LiveValue.lrActualPosition - T_Station_Work.THWWorkStation.TCtrlWork.rLastOverLimitPosition;
				END_IF;
				T_Station_Work.THWWorkStation.TCtrlWork.rLastOverLimitPosition:=ptrTAxisZ^.T_LiveValue.lrActualPosition;
				rStFct_TmpDiffOverLimitPosition:=T_Station_Work.THWWorkStation.TCtrlWork.rLastOverLimitPosition;
				IF (wStFct_Status = 1) OR (wStFct_Status = 3) THEN
					T_Station_Work.THWWorkStation.TCtrlWork.iOverLimitCounter:=T_Station_Work.THWWorkStation.TCtrlWork.iOverLimitCounter + 1;
				END_IF;
				IF (wStFct_Status = 2) OR (wStFct_Status = 3) THEN
					T_Station_Work.THWWorkStation.TCtrlWork.iOverLimitCounterTorque:=T_Station_Work.THWWorkStation.TCtrlWork.iOverLimitCounterTorque + 1;
				END_IF;
				IF (wStFct_Status = 4) THEN
					T_Station_Work.THWWorkStation.TCtrlWork.iOverLimitCounterSpeed:=T_Station_Work.THWWorkStation.TCtrlWork.iOverLimitCounterSpeed + 1;
				END_IF;
			END_IF;
			xStFct_ForceHC:=FALSE;
			(* init. variable *)
			xStFct_StopSlide:=FALSE;
			IF (T_Station_Parameter.T_StProcess.iWorkControlType <= 1) THEN
				iStFct_StepPrc:=iStFct_StepPrc + 1;
			ELSE
				rStFct_StopPosition:=LREAL_TO_REAL(ptrTAxisZ^.T_LiveValue.lrActualPosition);
				iStFct_StepPrc:=40;
			END_IF;
			xStFct_InitStep:=FALSE;
			RETURN;
		END_IF;
		IF (T_Station_Parameter.T_StProcess.iWorkControlType <= 1) THEN
			IF NOT(ptrTAxisZ^.T_CtrleSingle.xExecute) AND ptrTAxisZ^.T_CtrleSingle.xDone THEN
				IF NOT(gxProcessCylindricalAreaActive) OR xEndPosReachZylindricalProcess THEN
					(* Endposition erreicht-->Ausfunkprozedur starten *)
					T_Station_Work.TCtrlOnlineChange.xLockChange_Z_WorkSpeedForward:=TRUE;
					xStFct_StopSlide:=FALSE;
					xStFct_InitStep:=FALSE;
					IF T_Station_Parameter.T_StProcess.iSparkOutController<=2 THEN
						iStFct_StepPrc:=9; (* Use standard spark out with or without controller 1 *)
					ELSE
						iStFct_StepPrc:=50; (* Use spark out with fast controller 3 *)
					END_IF
				ELSE
					(* Beim neuen Ablauf darf die Max Endposition nicht erreicht werden *)
					xStFct_StopSlide:=FALSE;
					iStFct_StepPrc:=90;
					xStFct_InitStep:=FALSE;
				END_IF;
			END_IF;
		ELSE
			IF ((ptrTAxisZ^.T_LiveValue.lrActualPosition >= garPositionEndProcCalc[1]) AND NOT(gxProcessCylindricalAreaActive)) OR (xEndPosReachZylindricalProcess AND gxProcessCylindricalAreaActive) THEN
				xStFct_StartMainPrc:=FALSE;
				xStFct_InitStep:=FALSE;
				iStFct_StepPrc:=30; (* Reset Z axis in no matter what controller is selected for spark out -> make sure the axis is stationary *)
			END_IF;
		END_IF;
	4:	(* Abwarten bis die HubAchse stillsteht *)
		IF NOT(ptrTAxisZ^.T_CtrleSingle.xExecute) AND ptrTAxisZ^.T_CtrleSingle.xDone THEN
			(* init. variable *)
			rStFct_StopPosition:=ptrTAxisZ^.T_LiveValue.lrActualPosition;
			xStFct_StartMainPrc:=FALSE;
			xStFct_InitStep:=FALSE;
			iStFct_StepPrc:=iStFct_StepPrc + 1;
		END_IF;
	5:	(* HubAchse zurück auf StartPos setzen um den Rückwärts-Offset abzufahren *)
		ptrTAxisZ^.T_CtrleSingle.iFunction:=7;
		ptrTAxisZ^.T_CtrleSingle.lrPosition:=grZ_WorkStartPos;
		ptrTAxisZ^.T_CtrleSingle.lrVelocity:=T_Station_Parameter.T_OnlineChange.rWorkingSpeedBackward;
		ptrTAxisZ^.T_CtrleSingle.xExecute:=TRUE;
		iStFct_StepPrc:=iStFct_StepPrc + 1;
	6:	(* HubAchse fährt mindestens den Rückwärts-Offset zurück und wird gestoppt sobald die HC Sensoren nicht mehr bedämpft sind *)
		T_Station_Work.TCtrlOnlineChange.xLockChange_Z_WorkSpeedBackward:=ptrTAxisZ^.T_CtrleSingle.xNotMoving;
		IF ptrTAxisZ^.T_LiveValue.lrActualPosition < (rStFct_StopPosition + T_Station_Parameter.T_OnlineChange.rWorkingOffsetBackward) THEN
			IF NOT(xStFct_ToolDeflectionActiv) AND NOT(ptrTCylToolTorqueHC^.T_CtrleCyl.xStatePosOn) AND NOT(ptrTSensorTorque^.T_CtrleCyl.xStatePosOn) THEN
				xStFct_StopSlide:=TRUE;
			END_IF;
			IF xStFct_StopSlide AND NOT(ptrTAxisZ^.T_CtrleSingle.xExecute) AND NOT(ptrTAxisZ^.T_CtrleSingle.xDone) AND
			    NOT(ptrTAxisZ^.T_CtrleSingle.xNotMoving) AND (ptrTAxisZ^.T_CtrleSingle.iFunction <> 12) THEN
				T_Station_Work.TCtrlOnlineChange.xLockChange_Z_WorkSpeedBackward:=TRUE;
				ptrTAxisZ^.T_CtrleSingle.iFunction:=5;
				ptrTAxisZ^.T_CtrleSingle.xExecute:=TRUE;
				(* init. variable *)
				xStFct_StopSlide:=FALSE;
				iStFct_StepPrc:=iStFct_StepPrc + 1;
				RETURN;
			END_IF
		END_IF;
		IF NOT(ptrTAxisZ^.T_CtrleSingle.xExecute) AND ptrTAxisZ^.T_CtrleSingle.xDone THEN
			T_Station_Work.TCtrlOnlineChange.xLockChange_Z_WorkSpeedBackward:=TRUE;
			IF (iStFct_TmpHCStartPosCounter >= T_Station_Parameter.T_StProcess.iHCStartProcPosCounter) THEN	(* Counter bestimmt wie oft die Startposition erreicht werden darf, bis der Prozess abgebrochen wird *)
			(* end *)
				T_Station_Work.THWWorkStation.TCtrlWork.xWorkingFinished:=TRUE;
				(* Startposition mit max Anzahl zu erreichender StartPosition erreicht-->Prozess abgebrochen-->NoGo Part *)
				T_Station_Work.THWWorkStation.TCtrlWork.bPartQuality:=5;	(* < niO kein Einf. > *)
				xStFct_StartMainPrc:=FALSE;
				xStFct_InitStep:=FALSE;
				iStFct_StepPrc:=12;	(* Hubachse wieder auf LadePos setzen *)
			ELSE
				iStFct_TmpHCStartPosCounter:=iStFct_TmpHCStartPosCounter + 1;
				(* init. variable *)
				iStFct_StepPrc:=iStFct_StepPrc + 1;	(* HubAchse hat StartPosition erreicht, Vorwärtsbewegung muss wieder aktiviert werden *)
			END_IF;
		END_IF
	7:	(* Abwarten bis Achse gestoppt hat *)
		IF NOT(ptrTAxisZ^.T_CtrleSingle.xExecute) AND ptrTAxisZ^.T_CtrleSingle.xDone THEN
			xStFct_InitStep:=FALSE;
			iStFct_StepPrc:=iStFct_StepPrc + 1;
		END_IF
	8:	(* Vorwärtsbewegung wieder starten *)
		IF NOT(xStFct_InitStep) THEN
			xStFct_InitStep:=TRUE;
			ptrTAxisZ^.T_CtrleSingle.iFunction:=7;	(* Absolut Bewegung *)
			IF NOT(gxProcessCylindricalAreaActive) THEN
				ptrTAxisZ^.T_CtrleSingle.lrPosition:=garPositionEndProcCalc[1];	(* AxisSlide auf EndPosition setzen *)
			ELSE
				(* Das ist der neue Ablauf wo man einen Zylindrische Position definieren kann und aber dieser Position wenn das Drehmoment einem definierten Schwellwert unterschritten wird, dann ist dies das Prozessende. Wird aber diese unten übergebene Position erreicht, dann wertet es als Fehler *)
				ptrTAxisZ^.T_CtrleSingle.lrPosition:=T_Station_Parameter.T_StProcess.rPositionEndProcMaxInc;
			END_IF;
			ptrTAxisZ^.T_CtrleSingle.lrVelocity:=T_Station_Parameter.T_OnlineChange.rWorkingSpeedForward;
			ptrTAxisZ^.T_CtrleSingle.xExecute:=TRUE;
		END_IF;
		IF NOT(ptrTAxisZ^.T_CtrleSingle.xExecute) AND NOT(ptrTAxisZ^.T_CtrleSingle.xNotMoving) AND NOT(ptrTAxisZ^.T_CtrleSingle.xDone) THEN
			xStFct_StartMainPrc:=FALSE;
			xStFct_InitStep:=FALSE;
			iStFct_StepPrc:=3;
		END_IF;
	9:	(* Ausfunken starten *)
		IF NOT(xStFct_InitStep) THEN
			xStFct_InitStep:=TRUE;
			xStFct_StartSparkOutProcess:=TRUE;
			T_Station_Work.TCtrlOnlineChange.xLockChange_S_WorkSpindleSpeed:=TRUE;
			T_Station_Work.TCtrlOnlineChange.xLockChangeCylToolDeflectionForce:=TRUE;
			T_Station_Work.TCtrlOnlineChange.xLockChangeCylToolTorqueLevel:=TRUE;
			T_Station_Work.THWWorkStation.TCtrlWork.xSparkOutActive:=TRUE;
		END_IF;
		IF NOT(xStFct_StartSparkOutProcess) AND fbStFct_SparkOutProcess.xEnd AND NOT(fbStFct_SparkOutProcess.xBlockProcess) AND NOT(fbStFct_SparkOutProcess.xRepeatProcess) THEN
			xStFct_SparkOutDone:=TRUE;
			T_Station_Work.THWWorkStation.TCtrlWork.xSparkOutActive:=FALSE;
			T_Station_Work.TCtrlOnlineChange.xLockChange_S_WorkSpindleSpeed:=TRUE;
			T_Station_Work.TCtrlOnlineChange.xLockChangeCylToolDeflectionForce:=FALSE;
			T_Station_Work.TCtrlOnlineChange.xLockChangeCylToolTorqueLevel:=FALSE;
			IF ((T_Station_Parameter.T_OnlineChange.rWorkingSpindleSpeed > 0) AND (T_Station_Parameter.T_StProcess.rOutfeedSpindleSpeed < 0))
			OR ((T_Station_Parameter.T_OnlineChange.rWorkingSpindleSpeed < 0) AND (T_Station_Parameter.T_StProcess.rOutfeedSpindleSpeed > 0)) THEN
			(*IF (T_Station_Parameter.T_StProcess.rOutfeedSpindleSpeed > 0) THEN	*)	(* IGS1 neu mit umgekehrter Geschwindigkeit ausfahren zuerst Spindel stoppen, geht nicht anders, mit Dave besprochen *)
				iStFct_StepPrc:=20;
			ELSE
				IF T_Station_Parameter.T_StProcess.iOutfeedStrokeController <=2 THEN
					iStFct_StepPrc:=10; (* Standard outfeed stroke with or without controller 1 *)
				ELSE
					iStFct_StepPrc:=60; (* Outfeed stroke with fast control *)
				END_IF
			END_IF;
			xStFct_InitStep:=FALSE;
			RETURN;
		END_IF;
		IF NOT(xStFct_StartSparkOutProcess) AND fbStFct_SparkOutProcess.xEnd AND fbStFct_SparkOutProcess.xRepeatProcess THEN
			T_Station_Work.THWWorkStation.TCtrlWork.xSparkOutActive:=FALSE;
			T_Station_Work.TCtrlOnlineChange.xLockChangeCylToolDeflectionForce:=FALSE;
			T_Station_Work.TCtrlOnlineChange.xLockChangeCylToolTorqueLevel:=FALSE;
			wStFct_Status:=fbStFct_SparkOutProcess.wStatus;
			IF (rStFct_TmpDiffOverLimitPosition <> 0) THEN
				T_Station_Work.THWWorkStation.TCtrlWork.rDiffOverLimitPosition:=ptrTAxisZ^.T_LiveValue.lrActualPosition - T_Station_Work.THWWorkStation.TCtrlWork.rLastOverLimitPosition;
			END_IF;
			rStFct_SetZHCPosition:=fbStFct_SparkOutProcess.rLastOverLimitPosition;
			T_Station_Work.THWWorkStation.TCtrlWork.rLastOverLimitPosition:=fbStFct_SparkOutProcess.rLastOverLimitPosition;
			rStFct_TmpDiffOverLimitPosition:=T_Station_Work.THWWorkStation.TCtrlWork.rLastOverLimitPosition;
			T_Station_Work.THWWorkStation.TCtrlWork.xDeflectionLastHC:=FALSE;
			T_Station_Work.THWWorkStation.TCtrlWork.xTorqueLastHC:=FALSE;
			IF (wStFct_Status = 1) OR (wStFct_Status = 3) THEN
				T_Station_Work.THWWorkStation.TCtrlWork.iOverLimitCounter:=T_Station_Work.THWWorkStation.TCtrlWork.iOverLimitCounter + 1;
				T_Station_Work.THWWorkStation.TCtrlWork.xDeflectionLastHC:=TRUE;
			END_IF;
			IF (wStFct_Status = 2) OR (wStFct_Status = 3) THEN
				T_Station_Work.THWWorkStation.TCtrlWork.iOverLimitCounterTorque:=T_Station_Work.THWWorkStation.TCtrlWork.iOverLimitCounterTorque + 1;
				T_Station_Work.THWWorkStation.TCtrlWork.xTorqueLastHC:=TRUE;
			END_IF;
			iStFct_StepPrc:=4;
			xStFct_InitStep:=FALSE;
		END_IF;
	10:	(* Prozess beendet, HubAchse kann wieder auf LadePosition gesetzt *)
		IF (T_Station_Parameter.T_StProcess.rZ1AxisPosSwitchOAxisOff >= garPositionEndProcCalc[1])
		OR ((ptrTAxisZ^.T_LiveValue.lrActualPosition <= T_Station_Parameter.T_StProcess.rZ1AxisPosSwitchOAxisOff)
		OR (ABS(ptrTAxisZ^.T_LiveValue.lrActualPosition - T_Station_Parameter.T_StProcess.rPositionLoad) <= 10.0)) THEN
			QxFastStrokeOn_St1:=FALSE;
		END_IF;
		IF NOT(xStFct_InitStep) THEN
			xStFct_InitStep:=TRUE;
			xStFct_OutfeedStrokeRunning:=TRUE;
			T_Station_Work.THWWorkStation.TCtrlWork.xWorkingFinished:=TRUE;
			(* Auswertung der Qualität des Teiles *)
			IF NOT(xStFct_MinTimeProcessReady) THEN
				(* Prozess hat Mindest Zeit nicht überschritten *)
				T_Station_Work.THWWorkStation.TCtrlWork.bPartQuality:=3;	(* < niO min Zeit > *)
			ELSIF (T_Station_Work.THWWorkStation.TCtrlWork.iOverLimitCounter = 0) AND (T_Station_Work.THWWorkStation.TCtrlWork.iOverLimitCounterTorque = 0) THEN
				(* Bearbeitungsprozess hatte keinen Ausschlag, MindestZeit wurde aber überschritten *)
				T_Station_Work.THWWorkStation.TCtrlWork.bPartQuality:=2;	(* < iO kein HC > *)
				IF T_Station_Parameter.T_StProcess.xPositionEndProcIncOnOff THEN
					garPositionEndProcCalc[1]:=garPositionEndProcCalc[1] + T_Station_Parameter.T_StProcess.rPositionEndProInc;	(* EndPos Inkrementieren *)
				END_IF;
			ELSIF (T_Station_Work.THWWorkStation.TCtrlWork.iOverLimitCounter <> 0) OR (T_Station_Work.THWWorkStation.TCtrlWork.iOverLimitCounterTorque <> 0) THEN
				(* Bearbeitungsprozess hatte mindestens einen Ausschlag, MindestZeit wurde aber überschritten *)
				T_Station_Work.THWWorkStation.TCtrlWork.bPartQuality:=1;	(* < iO HC > *)
				IF T_Station_Parameter.T_StProcess.xPositionEndProcIncOnOff THEN
					garPositionEndProcCalc[1]:=garPositionEndProcCalc[1] + T_Station_Parameter.T_StProcess.rPositionEndProInc;	(* EndPos Inkrementieren *)
				END_IF;
			END_IF;
			ptrTAxisZ^.T_CtrleSingle.iFunction:=7;	(* Absolut Bewegung *)
			ptrTAxisZ^.T_CtrleSingle.lrPosition:=grZ_LoadPos;	(* AxisSlide auf BearbStartPosition setzen *)
			ptrTAxisZ^.T_CtrleSingle.lrVelocity:=rOutfeedStrokeAxisSpeed;
			ptrTAxisZ^.T_CtrleSingle.xExecute:=TRUE;
			(* Spindel mit Ausfahrgeschwindigkeit *)
			IF ptrTAxisS^.T_CtrleSingle.xNotMoving THEN
				ptrTAxisS^.T_CtrleSingle.iFunction:=6;	(* Move Velocity *)
			ELSE
				ptrTAxisS^.T_CtrleSingle.iFunction:=12;	(* Move Velocity *)
			END_IF;
			ptrTAxisS^.T_CtrleSingle.lrVelocity:=T_Station_Parameter.T_StProcess.rOutfeedSpindleSpeed;
			ptrTAxisS^.T_CtrleSingle.xExecute:=TRUE;
			IF NOT(ptrTAxisBubbler^.T_CtrleDCAxis.xNotMoving) THEN
				(* Abstreifer ZU *)
				QxCylStripperClose_St1:=TRUE;
				QxCylStripperOpen_St1:=FALSE;
			END_IF
		END_IF;
		IF NOT(ptrTAxisZ^.T_CtrleSingle.xExecute) AND ptrTAxisZ^.T_CtrleSingle.xDone AND
		     NOT(ptrTAxisS^.T_CtrleSingle.xExecute) AND ptrTAxisS^.T_CtrleSingle.xDone THEN
			xStFct_StartMainPrc:=FALSE;
			xStFct_InitStep:=FALSE;
			iStFct_StepPrc:=iStFct_StepPrc + 1;
		END_IF;
	11:	(* Prozess beendet, HubAchse kann wieder auf LadePosition gesetzt *)
		IF NOT(xStFct_InitStep) THEN
			xStFct_InitStep:=TRUE;
			xStFct_OutfeedStrokeRunning:=FALSE;
			ptrTAxisZ^.T_CtrleSingle.iFunction:=7;	(* Absolut Bewegung *)
			ptrTAxisZ^.T_CtrleSingle.lrPosition:=grZ_LoadPos;	(* AxisSlide auf LadePosition setzen *)
			ptrTAxisZ^.T_CtrleSingle.lrVelocity:=rOutfeedStrokeAxisSpeed;
			ptrTAxisZ^.T_CtrleSingle.xExecute:=TRUE;
			IF NOT(ptrTAxisBubbler^.T_CtrleDCAxis.xNotMoving) THEN
				(* Abstreifer ZU *)
				QxCylStripperClose_St1:=TRUE;
				QxCylStripperOpen_St1:=FALSE;
			END_IF
		END_IF;
		IF NOT(ptrTAxisZ^.T_CtrleSingle.xExecute) AND ptrTAxisZ^.T_CtrleSingle.xDone THEN
			xStFct_StartMainPrc:=FALSE;
			xStFct_InitStep:=FALSE;
			iStFct_StepPrc:=0;
			xStFct_SetEnd:=TRUE;
			IF xProcessDone THEN
				IF (NOT(ptrTAxisS^.T_CtrleSingle.xNotMoving) OR NOT(ptrTAxisS^.T_CtrleSingle.xDone)) AND
				     NOT((ptrTAxisS^.T_CtrleSingle.iFunction = 5) AND NOT(ptrTAxisS^.T_CtrleSingle.xDone)) AND NOT(ptrTAxisS^.T_CtrleSingle.xErr) THEN
					ptrTAxisS^.T_CtrleSingle.iFunction:=5;
					ptrTAxisS^.T_CtrleSingle.xExecute:=TRUE;
				END_IF;
			END_IF;
			(* Abstreifer AUF *)
			QxCylStripperClose_St1:=FALSE;
			QxCylStripperOpen_St1:=TRUE;
		END_IF;
	12:	(* Bei max. erreicht Startposition-->HubAchse wieder auf LadePosition gesetzt *)
		IF (T_Station_Parameter.T_StProcess.rZ1AxisPosSwitchOAxisOff >= garPositionEndProcCalc[1])
		OR ((ptrTAxisZ^.T_LiveValue.lrActualPosition <= T_Station_Parameter.T_StProcess.rZ1AxisPosSwitchOAxisOff)
		OR (ABS(ptrTAxisZ^.T_LiveValue.lrActualPosition - T_Station_Parameter.T_StProcess.rPositionLoad) <= 10.0)) THEN
			QxFastStrokeOn_St1:=FALSE;
		END_IF;
		IF NOT(xStFct_InitStep) THEN
			xStFct_InitStep:=TRUE;
			ptrTAxisZ^.T_CtrleSingle.iFunction:=7;	(* Absolut Bewegung *)
			ptrTAxisZ^.T_CtrleSingle.lrPosition:=grZ_LoadPos;	(* AxisSlide auf BearbStartPosition setzen *)
			ptrTAxisZ^.T_CtrleSingle.lrVelocity:=rOutfeedStrokeAxisSpeed;
			ptrTAxisZ^.T_CtrleSingle.xExecute:=TRUE;
			(* Spindel mit Ausfahrgeschwindigkeit *)
			IF ptrTAxisS^.T_CtrleSingle.xNotMoving THEN
				ptrTAxisS^.T_CtrleSingle.iFunction:=6;	(* Move Velocity *)
			ELSE
				ptrTAxisS^.T_CtrleSingle.iFunction:=12;	(* Move Velocity *)
			END_IF;
			ptrTAxisS^.T_CtrleSingle.lrVelocity:=T_Station_Parameter.T_StProcess.rOutfeedSpindleSpeed;
			ptrTAxisS^.T_CtrleSingle.xExecute:=TRUE;
			IF NOT(ptrTAxisBubbler^.T_CtrleDCAxis.xNotMoving) THEN
				(* Abstreifer ZU *)
				QxCylStripperClose_St1:=TRUE;
				QxCylStripperOpen_St1:=FALSE;
			END_IF
		END_IF;
		IF NOT(ptrTAxisZ^.T_CtrleSingle.xExecute) AND ptrTAxisZ^.T_CtrleSingle.xDone AND
		     NOT(ptrTAxisS^.T_CtrleSingle.xExecute) AND ptrTAxisS^.T_CtrleSingle.xDone THEN
			xStFct_StartMainPrc:=FALSE;
			xStFct_InitStep:=FALSE;
			iStFct_StepPrc:=iStFct_StepPrc + 1;
		END_IF;
	13:	(* Bei max. erreicht Startposition-->HubAchse wieder auf LadePosition gesetzt *)
		IF NOT(xStFct_InitStep) THEN
			xStFct_InitStep:=TRUE;
			ptrTAxisZ^.T_CtrleSingle.iFunction:=7;	(* Absolut Bewegung *)
			ptrTAxisZ^.T_CtrleSingle.lrPosition:=grZ_LoadPos;	(* AxisSlide auf LadePosition setzen *)
			ptrTAxisZ^.T_CtrleSingle.lrVelocity:=rOutfeedStrokeAxisSpeed;
			ptrTAxisZ^.T_CtrleSingle.xExecute:=TRUE;
			IF NOT(ptrTAxisBubbler^.T_CtrleDCAxis.xNotMoving) THEN
				(* Abstreifer ZU *)
				QxCylStripperClose_St1:=TRUE;
				QxCylStripperOpen_St1:=FALSE;
			END_IF
		END_IF;
		IF NOT(ptrTAxisZ^.T_CtrleSingle.xExecute) AND ptrTAxisZ^.T_CtrleSingle.xDone THEN
			xStFct_StartMainPrc:=FALSE;
			xStFct_InitStep:=FALSE;
			iStFct_StepPrc:=0;
			xStFct_SetEnd:=TRUE;
			IF xProcessDone THEN
				IF (NOT(ptrTAxisS^.T_CtrleSingle.xNotMoving) OR NOT(ptrTAxisS^.T_CtrleSingle.xDone)) AND
				     NOT((ptrTAxisS^.T_CtrleSingle.iFunction = 5) AND NOT(ptrTAxisS^.T_CtrleSingle.xDone)) AND NOT(ptrTAxisS^.T_CtrleSingle.xErr) THEN
					ptrTAxisS^.T_CtrleSingle.iFunction:=5;
					ptrTAxisS^.T_CtrleSingle.xExecute:=TRUE;
				END_IF;
			END_IF;
			(* Abstreifer AUF *)
			QxCylStripperClose_St1:=FALSE;
			QxCylStripperOpen_St1:=TRUE;
		END_IF;
	(* Gilt nur für falls HW ausgeschaltet ist *)
	14:	IF NOT(xStFct_InitStep) THEN
			xStFct_InitStep:=TRUE;
			TONWorkTime(IN:=FALSE);
		END_IF;
		TONWorkTime(IN:=TRUE,PT:=T#3s);
		IF TONWorkTime.Q THEN
			TONWorkTime(IN:=FALSE);
			xStFct_StartMainPrc:=FALSE;
			xStFct_InitStep:=FALSE;
			iStFct_StepPrc:=iStFct_StepPrc + 1;
			T_Station_Work.THWWorkStation.TCtrlWork.xWorkingFinished:=TRUE;
			(* Bearbeitungsprozess hatte keinen Ausschlag, MindestZeit wurde aber überschritten *)
			T_Station_Work.THWWorkStation.TCtrlWork.bPartQuality:=2;	(* < iO kein HC > *)
			IF T_Station_Parameter.T_StProcess.xPositionEndProcIncOnOff THEN
				garPositionEndProcCalc[1]:=garPositionEndProcCalc[1] + T_Station_Parameter.T_StProcess.rPositionEndProInc;
			END_IF;
		END_IF;
	(* Gilt nur für falls HW ausgeschaltet ist *)
	15:	IF NOT(xStFct_InitStep) THEN
			xStFct_InitStep:=TRUE;
			TONWorkTime(IN:=FALSE);
		END_IF;
		TONWorkTime(IN:=TRUE,PT:=T#2s);
		IF TONWorkTime.Q THEN
			TONWorkTime(IN:=FALSE);
			wStFct_Status:=0;
			xStFct_StartMainPrc:=FALSE;
			xStFct_InitStep:=FALSE;
			iStFct_StepPrc:=0;
			xStFct_SetEnd:=TRUE;
		END_IF;


	20:	(* Spindel stoppen *)	(* IGS1 neu mit umgekehrter Geschwindigkeit ausfahren, mit YGD besprochen *)
		IF NOT(xStFct_InitStep) THEN
			xStFct_InitStep:=TRUE;
			ptrTAxisS^.T_CtrleSingle.iFunction:=5;
			ptrTAxisS^.T_CtrleSingle.xExecute:=TRUE;
		END_IF;
		IF NOT(ptrTAxisS^.T_CtrleSingle.xExecute) AND ptrTAxisS^.T_CtrleSingle.xDone THEN
			xStFct_StartMainPrc:=FALSE;
			xStFct_InitStep:=FALSE;
			IF T_Station_Parameter.T_StProcess.iOutfeedStrokeController <=2 AND T_Station_Parameter.T_StProcess.iSparkOutController = 3 THEN
				iStFct_StepPrc:=30; (* Z axis need to be reset if coming from fast control and go to position control *)
			ELSIF T_Station_Parameter.T_StProcess.iOutfeedStrokeController <=2 THEN
				iStFct_StepPrc:=10; (* Standard outfeed stroke with or without controller 1 *)
			ELSE
				iStFct_StepPrc:=60; (* Outfeed stroke with fast control *)
			END_IF
		END_IF;

	30:	(* Bei Drehzahlregler passt der Sollwert der Position nicht mehr mit dem Ist Wert und deshalb muss ein Reset durchgeführt werden *)
		IF NOT(xStFct_InitStep) THEN
			xStFct_InitStep:=TRUE;
			ptrTAxisZ^.T_CtrleSingle.iFunction:=1;
			ptrTAxisZ^.T_CtrleSingle.xExecute:=TRUE;
		END_IF;
		IF NOT(ptrTAxisZ^.T_CtrleSingle.xExecute) AND ptrTAxisZ^.T_CtrleSingle.xDone THEN
			xStFct_StartMainPrc:=FALSE;
			xStFct_InitStep:=FALSE;
			iStFct_StepPrc:=iStFct_StepPrc + 1;
		END_IF;
	31:	(* Bei Drehzahlregler ohne verweilzeit und man dann direkt eine Positionsfahrt auslösen will, dann führt es zum Fehler 18000 der Achse *)
		IF NOT(xStFct_InitStep) THEN
			xStFct_InitStep:=TRUE;
			TONWaitMovement(IN:=FALSE);
		END_IF;
		TONWaitMovement(IN:=TRUE,PT:=T#0.3s);
		IF TONWaitMovement.Q THEN
			TONWaitMovement(IN:=FALSE);
			xStFct_StartMainPrc:=FALSE;
			xStFct_InitStep:=FALSE;
			IF gxProcessCylindricalAreaActive AND NOT(xEndPosReachZylindricalProcess) THEN
				(* Beim neuen Ablauf darf die Max Endposition nicht erreicht werden *)
				iStFct_StepPrc:=90;
			ELSE
				IF NOT(xStFct_SparkOutDone) AND T_Station_Parameter.T_StProcess.iSparkOutController <= 2 THEN
					iStFct_StepPrc:=9; 		(* Use standard spark out with or without controller 1 *)
				ELSIF NOT(xStFct_SparkOutDone) AND T_Station_Parameter.T_StProcess.iSparkOutController = 3 THEN
					iStFct_StepPrc:=50; 	(* Use spark out with fast controller 3 *)
				ELSIF T_Station_Parameter.T_StProcess.iOutfeedStrokeController <= 2 THEN
					iStFct_StepPrc:=10;	 (* Use standard outfeed stroke  with or without controller 1 *)
				ELSE
					iStFct_StepPrc:=60;	 (* Use outfeed stroke with fast controller 3 *)
				END_IF
			END_IF;
		END_IF;

	(* Beim Drehzahlregler wenn ein HC eintrifft für den Offset zurück wird auch mit dem Drehzahlregler bewegt, anderenfalls müsste man die Achse resetten *)
	40:	IF (T_Station_Parameter.T_StProcess.iWorkControlType = 2) THEN
			rStFct_CalcZSpeed:=(ABS(T_Station_Parameter.T_StProcess.rZ_PID_MinSpeed)/100.0) * BYTE_TO_REAL(T_ExchgParam.byOverride);
		ELSE
			rStFct_CalcZSpeed:=(T_Station_Parameter.T_OnlineChange.rWorkingSpeedBackward/100.0) * BYTE_TO_REAL(T_ExchgParam.byOverride);
		END_IF;
		T_Z_St1_Ctrle.diVelocityCommandValue:=LREAL_TO_DINT(rStFct_CalcZSpeed * 558349.25) ; (* 11166985 --> 20mm/s --> 1mm/s = 558349.25 *)
		T_Station_Work.TCtrlOnlineChange.xLockChange_Z_WorkSpeedBackward:=ptrTAxisZ^.T_CtrleSingle.xNotMoving;
		IF ptrTAxisZ^.T_LiveValue.lrActualPosition < (rStFct_StopPosition + T_Station_Parameter.T_OnlineChange.rWorkingOffsetBackward) THEN
			IF NOT(xStFct_ToolDeflectionActiv) AND NOT(ptrTSensorTorque^.T_CtrleCyl.xStatePosOn) THEN
				T_Z_St1_Ctrle.diVelocityCommandValue:=0;
				xStFct_StartMainPrc:=FALSE;
				xStFct_InitStep:=FALSE;
				iStFct_StepPrc:=3;
			END_IF;
		END_IF;

	50: 	(* Ausfunken mit schnellem Regler *)
		IF NOT(xStFct_InitStep) THEN
			xStFct_InitStep:=TRUE;
			xStFct_StartSparkOutProcess:=TRUE;
			T_Station_Work.TCtrlOnlineChange.xLockChange_S_WorkSpindleSpeed:=TRUE;
			T_Station_Work.TCtrlOnlineChange.xLockChangeCylToolDeflectionForce:=TRUE;
			T_Station_Work.TCtrlOnlineChange.xLockChangeCylToolTorqueLevel:=TRUE;
			T_Station_Work.THWWorkStation.TCtrlWork.xSparkOutActive:=TRUE;
		END_IF;
		IF NOT(xStFct_StartSparkOutProcess) AND NOT(xStFct_SparkOutRunning) AND NOT(xStFct_RepeatProcess) THEN
			xStFct_SparkOutDone:=TRUE;
			T_Z_St1_Ctrle.diVelocityCommandValue:=0; (* Make sure Z axis is not moving anymore *)
			T_Station_Work.THWWorkStation.TCtrlWork.xSparkOutActive:=FALSE;
			T_Station_Work.TCtrlOnlineChange.xLockChange_S_WorkSpindleSpeed:=TRUE;
			T_Station_Work.TCtrlOnlineChange.xLockChangeCylToolDeflectionForce:=FALSE;
			T_Station_Work.TCtrlOnlineChange.xLockChangeCylToolTorqueLevel:=FALSE;
			IF ((T_Station_Parameter.T_OnlineChange.rWorkingSpindleSpeed > 0) AND (T_Station_Parameter.T_StProcess.rOutfeedSpindleSpeed < 0))
			OR ((T_Station_Parameter.T_OnlineChange.rWorkingSpindleSpeed < 0) AND (T_Station_Parameter.T_StProcess.rOutfeedSpindleSpeed > 0)) THEN
			(*IF (T_Station_Parameter.T_StProcess.rOutfeedSpindleSpeed > 0) THEN	*)	(* IGS1 neu mit umgekehrter Geschwindigkeit ausfahren zuerst Spindel stoppen, geht nicht anders, mit Dave besprochen *)
				iStFct_StepPrc:=20;
			ELSE
				IF T_Station_Parameter.T_StProcess.iOutfeedStrokeController <= 2 THEN
					iStFct_StepPrc:=30; (* Reset Z axis *)
				ELSE
					iStFct_StepPrc:=60; (* Outfeed stroke with fast control *)
				END_IF;
			END_IF;
			xStFct_StartMainPrc:=FALSE;
			xStFct_InitStep:=FALSE;
			RETURN;
		END_IF;
		IF NOT(xStFct_StartSparkOutProcess) AND NOT(xStFct_SparkOutRunning) AND xStFct_RepeatProcess THEN
			T_Station_Work.THWWorkStation.TCtrlWork.xSparkOutActive:=FALSE;
			T_Station_Work.TCtrlOnlineChange.xLockChangeCylToolDeflectionForce:=FALSE;
			T_Station_Work.TCtrlOnlineChange.xLockChangeCylToolTorqueLevel:=FALSE;
			(*wStFct_Status:=fbStFct_SparkOutProcess.wStatus;*)

			(*IF (rStFct_TmpDiffOverLimitPosition <> 0) THEN
				T_Station_Work.THWWorkStation.TCtrlWork.rDiffOverLimitPosition:=ptrTAxisZ^.T_LiveValue.lrActualPosition - T_Station_Work.THWWorkStation.TCtrlWork.rLastOverLimitPosition;
			END_IF;
			rStFct_SetZHCPosition:=fbStFct_SparkOutProcess.rLastOverLimitPosition;
			T_Station_Work.THWWorkStation.TCtrlWork.rLastOverLimitPosition:=fbStFct_SparkOutProcess.rLastOverLimitPosition;
			rStFct_TmpDiffOverLimitPosition:=T_Station_Work.THWWorkStation.TCtrlWork.rLastOverLimitPosition;*)

			T_Station_Work.THWWorkStation.TCtrlWork.xDeflectionLastHC:=FALSE;
			T_Station_Work.THWWorkStation.TCtrlWork.xTorqueLastHC:=FALSE;
			IF (wStFct_Status = 1) OR (wStFct_Status = 3) THEN
				T_Station_Work.THWWorkStation.TCtrlWork.iOverLimitCounter:=T_Station_Work.THWWorkStation.TCtrlWork.iOverLimitCounter + 1;
				T_Station_Work.THWWorkStation.TCtrlWork.xDeflectionLastHC:=TRUE;
			END_IF;
			IF (wStFct_Status = 2) OR (wStFct_Status = 3) THEN
				T_Station_Work.THWWorkStation.TCtrlWork.iOverLimitCounterTorque:=T_Station_Work.THWWorkStation.TCtrlWork.iOverLimitCounterTorque + 1;
				T_Station_Work.THWWorkStation.TCtrlWork.xTorqueLastHC:=TRUE;
			END_IF;
			xStFct_StartMainPrc:=FALSE;
			xStFct_InitStep:=FALSE;
			iStFct_StepPrc:=40;
		END_IF;

	60: 	(* Rückfahrt Prozessende mit schnellem Regler *)
		IF (T_Station_Parameter.T_StProcess.rZ1AxisPosSwitchOAxisOff >= garPositionEndProcCalc[1])
		OR ((ptrTAxisZ^.T_LiveValue.lrActualPosition <= T_Station_Parameter.T_StProcess.rZ1AxisPosSwitchOAxisOff)
		OR (ABS(ptrTAxisZ^.T_LiveValue.lrActualPosition - T_Station_Parameter.T_StProcess.rPositionLoad) <= 10.0)) THEN
			QxFastStrokeOn_St1:=FALSE;
		END_IF;
		IF NOT(xStFct_InitStep) THEN
			xStFct_InitStep:=TRUE;
			xStFct_OutfeedStrokeRunning:=TRUE;
			T_Station_Work.THWWorkStation.TCtrlWork.xWorkingFinished:=TRUE;
			(* Auswertung der Qualität des Teiles *)
			IF NOT(xStFct_MinTimeProcessReady) THEN
				(* Prozess hat Mindest Zeit nicht überschritten *)
				T_Station_Work.THWWorkStation.TCtrlWork.bPartQuality:=3;	(* < niO min Zeit > *)
			ELSIF (T_Station_Work.THWWorkStation.TCtrlWork.iOverLimitCounter = 0) AND (T_Station_Work.THWWorkStation.TCtrlWork.iOverLimitCounterTorque = 0) THEN
				(* Bearbeitungsprozess hatte keinen Ausschlag, MindestZeit wurde aber überschritten *)
				T_Station_Work.THWWorkStation.TCtrlWork.bPartQuality:=2;	(* < iO kein HC > *)
				IF T_Station_Parameter.T_StProcess.xPositionEndProcIncOnOff THEN
					garPositionEndProcCalc[1]:=garPositionEndProcCalc[1] + T_Station_Parameter.T_StProcess.rPositionEndProInc;	(* EndPos Inkrementieren *)
				END_IF;
			ELSIF (T_Station_Work.THWWorkStation.TCtrlWork.iOverLimitCounter <> 0) OR (T_Station_Work.THWWorkStation.TCtrlWork.iOverLimitCounterTorque <> 0) THEN
				(* Bearbeitungsprozess hatte mindestens einen Ausschlag, MindestZeit wurde aber überschritten *)
				T_Station_Work.THWWorkStation.TCtrlWork.bPartQuality:=1;	(* < iO HC > *)
				IF T_Station_Parameter.T_StProcess.xPositionEndProcIncOnOff THEN
					garPositionEndProcCalc[1]:=garPositionEndProcCalc[1] + T_Station_Parameter.T_StProcess.rPositionEndProInc;	(* EndPos Inkrementieren *)
				END_IF;
			END_IF;

			rStFct_CtrlInputWorkingSpeed:=(-T_Station_Parameter.T_StProcess.rSpeedZAxisForBackward/100.0) * BYTE_TO_REAL(T_ExchgParam.byOverride);

